LIN {X 0,Y 509.297,Z 394.262,A -85,B 0,C 180,E1 -5484.06,E2 -5484.06} C_VEL
LIN {X 0,Y 509.19,Z 398.581,A -85,B 0,C 180,E1 -5485.25,E2 -5485.25} C_VEL
LIN {X 0,Y 509.246,Z 400.946,A -85,B 0,C 180,E1 -5486.043,E2 -5486.043} C_VEL
LIN {X 0,Y 509.201,Z 402.741,A -85,B 0,C 180,E1 -5486.835,E2 -5486.835} C_VEL
LIN {X 0,Y 509.113,Z 405.178,A -85,B 0,C 180,E1 -5488.418,E2 -5488.418} C_VEL
LIN {X 0,Y 509.076,Z 405.764,A -85,B 0,C 180,E1 -5489.209,E2 -5489.209} C_VEL
LIN {X 0,Y 509.076,Z 405.764,A -85,B 0,C 180,E1 -5490.791,E2 -5490.791} C_VEL
LIN {X 0,Y 509.113,Z 405.178,A -85,B 0,C 180,E1 -5491.582,E2 -5491.582} C_VEL
LIN {X 0,Y 509.201,Z 402.741,A -85,B 0,C 180,E1 -5493.165,E2 -5493.165} C_VEL
LIN {X 0,Y 509.206,Z 399.797,A -85,B 0,C 180,E1 -5494.353,E2 -5494.353} C_VEL
LIN {X 0,Y 509.283,Z 395.815,A -85,B 0,C 180,E1 -5495.543,E2 -5495.543} C_VEL
LIN {X 0,Y 509.305,Z 390.878,A -85,B 0,C 180,E1 -5496.696,E2 -5496.696} C_VEL
LIN {X 0,Y 509.461,Z 385.428,A -85,B 0,C 180,E1 -5497.73,E2 -5497.73} C_VEL
LIN {X 0,Y 509.641,Z 379.112,A -85,B 0,C 180,E1 -5498.725,E2 -5498.725} C_VEL
LIN {X 0,Y 509.831,Z 373.161,A -85,B 0,C 180,E1 -5499.521,E2 -5499.521} C_VEL
LIN {X 0,Y 509.999,Z 366.231,A -85,B 0,C 180,E1 -5500.32,E2 -5500.32} C_VEL
LIN {X 0,Y 510.309,Z 358.051,A -85,B 0,C 180,E1 -5501.117,E2 -5501.117} C_VEL
LIN {X 0,Y 510.555,Z 349.536,A -85,B 0,C 180,E1 -5501.815,E2 -5501.815} C_VEL
LIN {X 0,Y 510.838,Z 339.999,A -85,B 0,C 180,E1 -5502.464,E2 -5502.464} C_VEL
LIN {X 0,Y 511.107,Z 330.048,A -85,B 0,C 180,E1 -5503.012,E2 -5503.012} C_VEL
LIN {X 0,Y 511.372,Z 319.682,A -85,B 0,C 180,E1 -5503.461,E2 -5503.461} C_VEL
LIN {X 0,Y 511.591,Z 308.831,A -85,B 0,C 180,E1 -5503.809,E2 -5503.809} C_VEL
LIN {X 0,Y 511.838,Z 295.749,A -85,B 0,C 180,E1 -5504.081,E2 -5504.081} C_VEL
LIN {X 0,Y 512.093,Z 207.59,A -85,B 0,C 180,E1 -5505.325,E2 -5505.325} C_VEL
LIN {X 0,Y 510.014,Z 195.134,A -85,B 0,C 180,E1 -5505.587,E2 -5505.587} C_VEL
LIN {X 0,Y 510.036,Z 192.862,A -85,B 0,C 180,E1 -5505.997,E2 -5505.997} C_VEL
LIN {X 0,Y 510.351,Z 179.568,A -85,B 0,C 180,E1 -5508.673,E2 -5508.673} C_VEL
LIN {X 0,Y 510.701,Z 165.975,A -85,B 0,C 180,E1 -5511.388,E2 -5511.388} C_VEL
LIN {X 0,Y 511.205,Z 151.526,A -85,B 0,C 180,E1 -5514.358,E2 -5514.358} C_VEL
LIN {X 0,Y 510.606,Z 146.371,A -85,B 0,C 180,E1 -5515.475,E2 -5515.475} C_VEL
LIN {X 0,Y 509.929,Z 142.498,A -85,B 0,C 180,E1 -5516.381,E2 -5516.381} C_VEL
LIN {X 0,Y 509.875,Z 142.472,A -85,B 0,C 180,E1 -5518.844,E2 -5518.844} C_VEL
LIN {X 0,Y 509.822,Z 142.482,A -85,B 0,C 180,E1 -5521.59,E2 -5521.59} C_VEL
LIN {X 0,Y 509.848,Z 142.473,A -85,B 0,C 180,E1 -5524.413,E2 -5524.413} C_VEL
LIN {X 0,Y 509.818,Z 142.478,A -85,B 0,C 180,E1 -5527.34,E2 -5527.34} C_VEL
LIN {X 0,Y 509.838,Z 142.466,A -85,B 0,C 180,E1 -5530.382,E2 -5530.382} C_VEL
LIN {X 0,Y 509.822,Z 142.477,A -85,B 0,C 180,E1 -5533.062,E2 -5533.062} C_VEL
LIN {X 0,Y 509.822,Z 142.48,A -85,B 0,C 180,E1 -5535.793,E2 -5535.793} C_VEL
LIN {X 0,Y 509.854,Z 142.471,A -85,B 0,C 180,E1 -5538.574,E2 -5538.574} C_VEL
LIN {X 0,Y 509.849,Z 142.475,A -85,B 0,C 180,E1 -5541.786,E2 -5541.786} C_VEL
LIN {X 0,Y 509.831,Z 142.473,A -85,B 0,C 180,E1 -5544.622,E2 -5544.622} C_VEL
LIN {X 0,Y 509.862,Z 142.475,A -85,B 0,C 180,E1 -5547.48,E2 -5547.48} C_VEL
LIN {X 0,Y 509.857,Z 142.47,A -85,B 0,C 180,E1 -5550.273,E2 -5550.273} C_VEL
LIN {X 0,Y 509.882,Z 142.466,A -85,B 0,C 180,E1 -5552.944,E2 -5552.944} C_VEL
LIN {X 0,Y 509.862,Z 142.471,A -85,B 0,C 180,E1 -5555.573,E2 -5555.573} C_VEL
LIN {X 0,Y 509.848,Z 142.474,A -85,B 0,C 180,E1 -5558.998,E2 -5558.998} C_VEL
LIN {X 0,Y 509.886,Z 142.458,A -85,B 0,C 180,E1 -5561.999,E2 -5561.999} C_VEL
LIN {X 0,Y 509.908,Z 142.471,A -85,B 0,C 180,E1 -5564.818,E2 -5564.818} C_VEL
LIN {X 0,Y 509.897,Z 142.464,A -85,B 0,C 180,E1 -5568.124,E2 -5568.124} C_VEL
LIN {X 0,Y 509.911,Z 142.457,A -85,B 0,C 180,E1 -5571.279,E2 -5571.279} C_VEL
LIN {X 0,Y 509.975,Z 142.454,A -85,B 0,C 180,E1 -5573.67,E2 -5573.67} C_VEL
LIN {X 0,Y 510.051,Z 142.444,A -85,B 0,C 180,E1 -5577.63,E2 -5577.63} C_VEL
LIN {X 0,Y 510.06,Z 142.44,A -85,B 0,C 180,E1 -5580.789,E2 -5580.789} C_VEL
LIN {X 0,Y 509.952,Z 142.457,A -85,B 0,C 180,E1 -5583.16,E2 -5583.16} C_VEL
LIN {X 0,Y 509.974,Z 142.46,A -85,B 0,C 180,E1 -5586.329,E2 -5586.329} C_VEL
LIN {X 0,Y 509.911,Z 142.456,A -85,B 0,C 180,E1 -5588.72,E2 -5588.72} C_VEL
LIN {X 0,Y 509.9,Z 142.465,A -85,B 0,C 180,E1 -5591.931,E2 -5591.931} C_VEL
LIN {X 0,Y 509.889,Z 142.467,A -85,B 0,C 180,E1 -5595.241,E2 -5595.241} C_VEL
LIN {X 0,Y 509.884,Z 142.464,A -85,B 0,C 180,E1 -5598.001,E2 -5598.001} C_VEL
LIN {X 0,Y 509.845,Z 142.468,A -85,B 0,C 180,E1 -5601.001,E2 -5601.001} C_VEL
LIN {X 0,Y 509.832,Z 142.479,A -85,B 0,C 180,E1 -5603.563,E2 -5603.563} C_VEL
LIN {X 0,Y 509.909,Z 142.458,A -85,B 0,C 180,E1 -5606.379,E2 -5606.379} C_VEL
LIN {X 0,Y 509.872,Z 142.465,A -85,B 0,C 180,E1 -5608.844,E2 -5608.844} C_VEL
LIN {X 0,Y 509.821,Z 142.482,A -85,B 0,C 180,E1 -5611.589,E2 -5611.589} C_VEL
LIN {X 0,Y 509.85,Z 142.464,A -85,B 0,C 180,E1 -5614.413,E2 -5614.413} C_VEL
LIN {X 0,Y 509.814,Z 142.483,A -85,B 0,C 180,E1 -5617.34,E2 -5617.34} C_VEL
LIN {X 0,Y 509.833,Z 142.469,A -85,B 0,C 180,E1 -5620.382,E2 -5620.382} C_VEL
LIN {X 0,Y 509.836,Z 142.479,A -85,B 0,C 180,E1 -5623.064,E2 -5623.064} C_VEL
LIN {X 0,Y 509.825,Z 142.469,A -85,B 0,C 180,E1 -5625.792,E2 -5625.792} C_VEL
LIN {X 0,Y 509.853,Z 142.457,A -85,B 0,C 180,E1 -5628.575,E2 -5628.575} C_VEL
LIN {X 0,Y 509.847,Z 142.473,A -85,B 0,C 180,E1 -5631.786,E2 -5631.786} C_VEL
LIN {X 0,Y 509.827,Z 142.471,A -85,B 0,C 180,E1 -5633.729,E2 -5633.729} C_VEL
LIN {X 0,Y 509.161,Z 142.556,A -85,B 0,C 180,E1 -5634.388,E2 -5634.388} C_VEL
LIN {X 0,Y 506.344,Z 142.91,A -85,B 0,C 180,E1 -5635.46,E2 -5635.46} C_VEL
LIN {X 0,Y 503.952,Z 143.211,A -85,B 0,C 180,E1 -5636.324,E2 -5636.324} C_VEL
LIN {X 0,Y 502.903,Z 143.341,A -85,B 0,C 180,E1 -5636.99,E2 -5636.99} C_VEL
LIN {X 0,Y 502.806,Z 143.351,A -85,B 0,C 180,E1 -5637.216,E2 -5637.216} C_VEL
LIN {X 0,Y 502.826,Z 143.344,A -85,B 0,C 180,E1 -5640.062,E2 -5640.062} C_VEL
LIN {X 0,Y 502.83,Z 143.351,A -85,B 0,C 180,E1 -5642.533,E2 -5642.533} C_VEL
LIN {X 0,Y 502.825,Z 143.349,A -85,B 0,C 180,E1 -5645.299,E2 -5645.299} C_VEL
LIN {X 0,Y 502.781,Z 143.354,A -85,B 0,C 180,E1 -5647.827,E2 -5647.827} C_VEL
LIN {X 0,Y 502.822,Z 143.355,A -85,B 0,C 180,E1 -5650.4,E2 -5650.4} C_VEL
LIN {X 0,Y 502.83,Z 143.35,A -85,B 0,C 180,E1 -5652.932,E2 -5652.932} C_VEL
LIN {X 0,Y 502.842,Z 143.347,A -85,B 0,C 180,E1 -5655.429,E2 -5655.429} C_VEL
LIN {X 0,Y 502.874,Z 143.346,A -85,B 0,C 180,E1 -5658.717,E2 -5658.717} C_VEL
LIN {X 0,Y 502.899,Z 143.344,A -85,B 0,C 180,E1 -5661.967,E2 -5661.967} C_VEL
LIN {X 0,Y 502.936,Z 143.34,A -85,B 0,C 180,E1 -5664.387,E2 -5664.387} C_VEL
LIN {X 0,Y 503.023,Z 143.327,A -85,B 0,C 180,E1 -5667.598,E2 -5667.598} C_VEL
LIN {X 0,Y 503.025,Z 143.33,A -85,B 0,C 180,E1 -5670,E2 -5670} C_VEL
LIN {X 0,Y 503.023,Z 143.327,A -85,B 0,C 180,E1 -5672.402,E2 -5672.402} C_VEL
LIN {X 0,Y 502.936,Z 143.34,A -85,B 0,C 180,E1 -5675.613,E2 -5675.613} C_VEL
LIN {X 0,Y 502.899,Z 143.344,A -85,B 0,C 180,E1 -5678.033,E2 -5678.033} C_VEL
LIN {X 0,Y 502.874,Z 143.346,A -85,B 0,C 180,E1 -5681.283,E2 -5681.283} C_VEL
LIN {X 0,Y 502.842,Z 143.347,A -85,B 0,C 180,E1 -5684.571,E2 -5684.571} C_VEL
LIN {X 0,Y 502.858,Z 143.348,A -85,B 0,C 180,E1 -5687.907,E2 -5687.907} C_VEL
LIN {X 0,Y 502.825,Z 143.349,A -85,B 0,C 180,E1 -5690.536,E2 -5690.536} C_VEL
LIN {X 0,Y 502.793,Z 143.356,A -85,B 0,C 180,E1 -5693.04,E2 -5693.04} C_VEL
LIN {X 0,Y 502.836,Z 143.35,A -85,B 0,C 180,E1 -5695.675,E2 -5695.675} C_VEL
LIN {X 0,Y 502.838,Z 143.344,A -85,B 0,C 180,E1 -5698.372,E2 -5698.372} C_VEL
LIN {X 0,Y 502.793,Z 143.355,A -85,B 0,C 180,E1 -5701.5,E2 -5701.5} C_VEL
LIN {X 0,Y 502.8,Z 143.343,A -85,B 0,C 180,E1 -5704.444,E2 -5704.444} C_VEL
LIN {X 0,Y 502.776,Z 143.36,A -85,B 0,C 180,E1 -5707.178,E2 -5707.178} C_VEL
LIN {X 0,Y 502.783,Z 143.348,A -85,B 0,C 180,E1 -5710.015,E2 -5710.015} C_VEL
LIN {X 0,Y 502.797,Z 143.334,A -85,B 0,C 180,E1 -5712.199,E2 -5712.199} C_VEL
LIN {X 0,Y 502.796,Z 143.351,A -85,B 0,C 180,E1 -5715.468,E2 -5715.468} C_VEL
LIN {X 0,Y 502.825,Z 143.346,A -85,B 0,C 180,E1 -5717.864,E2 -5717.864} C_VEL
LIN {X 0,Y 502.797,Z 143.354,A -85,B 0,C 180,E1 -5721.024,E2 -5721.024} C_VEL
LIN {X 0,Y 502.781,Z 143.355,A -85,B 0,C 180,E1 -5724.167,E2 -5724.167} C_VEL
LIN {X 0,Y 502.828,Z 143.347,A -85,B 0,C 180,E1 -5726.993,E2 -5726.993} C_VEL
LIN {X 0,Y 502.809,Z 143.353,A -85,B 0,C 180,E1 -5730.065,E2 -5730.065} C_VEL
LIN {X 0,Y 502.831,Z 143.343,A -85,B 0,C 180,E1 -5732.534,E2 -5732.534} C_VEL
LIN {X 0,Y 502.824,Z 143.346,A -85,B 0,C 180,E1 -5735.299,E2 -5735.299} C_VEL
LIN {X 0,Y 502.78,Z 143.356,A -85,B 0,C 180,E1 -5737.827,E2 -5737.827} C_VEL
LIN {X 0,Y 502.821,Z 143.34,A -85,B 0,C 180,E1 -5740.401,E2 -5740.401} C_VEL
LIN {X 0,Y 502.829,Z 143.343,A -85,B 0,C 180,E1 -5742.932,E2 -5742.932} C_VEL
LIN {X 0,Y 502.841,Z 143.346,A -85,B 0,C 180,E1 -5745.43,E2 -5745.43} C_VEL
LIN {X 0,Y 502.873,Z 143.333,A -85,B 0,C 180,E1 -5748.717,E2 -5748.717} C_VEL
LIN {X 0,Y 502.897,Z 143.339,A -85,B 0,C 180,E1 -5751.967,E2 -5751.967} C_VEL
LIN {X 0,Y 502.934,Z 143.334,A -85,B 0,C 180,E1 -5754.387,E2 -5754.387} C_VEL
LIN {X 0,Y 503.02,Z 143.325,A -85,B 0,C 180,E1 -5757.598,E2 -5757.598} C_VEL
LIN {X 0,Y 503.024,Z 143.315,A -85,B 0,C 180,E1 -5760,E2 -5760} C_VEL
LIN {X 0,Y 503.021,Z 143.319,A -85,B 0,C 180,E1 -5762.403,E2 -5762.403} C_VEL
LIN {X 0,Y 502.934,Z 143.338,A -85,B 0,C 180,E1 -5765.614,E2 -5765.614} C_VEL
LIN {X 0,Y 502.898,Z 143.331,A -85,B 0,C 180,E1 -5768.034,E2 -5768.034} C_VEL
LIN {X 0,Y 502.874,Z 143.338,A -85,B 0,C 180,E1 -5771.284,E2 -5771.284} C_VEL
LIN {X 0,Y 502.842,Z 143.344,A -85,B 0,C 180,E1 -5774.571,E2 -5774.571} C_VEL
LIN {X 0,Y 502.859,Z 143.333,A -85,B 0,C 180,E1 -5777.907,E2 -5777.907} C_VEL
LIN {X 0,Y 502.826,Z 143.342,A -85,B 0,C 180,E1 -5780.537,E2 -5780.537} C_VEL
LIN {X 0,Y 502.789,Z 143.358,A -85,B 0,C 180,E1 -5783.041,E2 -5783.041} C_VEL
LIN {X 0,Y 502.838,Z 143.339,A -85,B 0,C 180,E1 -5785.676,E2 -5785.676} C_VEL
LIN {X 0,Y 502.838,Z 143.341,A -85,B 0,C 180,E1 -5788.373,E2 -5788.373} C_VEL
LIN {X 0,Y 502.792,Z 143.351,A -85,B 0,C 180,E1 -5791.499,E2 -5791.499} C_VEL
LIN {X 0,Y 502.804,Z 143.344,A -85,B 0,C 180,E1 -5793.994,E2 -5793.994} C_VEL
LIN {X 0,Y 502.776,Z 143.355,A -85,B 0,C 180,E1 -5797.178,E2 -5797.178} C_VEL
LIN {X 0,Y 502.787,Z 143.35,A -85,B 0,C 180,E1 -5800.016,E2 -5800.016} C_VEL
LIN {X 0,Y 502.802,Z 143.353,A -85,B 0,C 180,E1 -5802.2,E2 -5802.2} C_VEL
LIN {X 0,Y 502.785,Z 143.351,A -85,B 0,C 180,E1 -5805.471,E2 -5805.471} C_VEL
LIN {X 0,Y 502.82,Z 143.341,A -85,B 0,C 180,E1 -5808.935,E2 -5808.935} C_VEL
LIN {X 0,Y 502.794,Z 143.355,A -85,B 0,C 180,E1 -5812.047,E2 -5812.047} C_VEL
LIN {X 0,Y 502.8,Z 143.349,A -85,B 0,C 180,E1 -5815.035,E2 -5815.035} C_VEL
LIN {X 0,Y 502.785,Z 143.354,A -85,B 0,C 180,E1 -5817.916,E2 -5817.916} C_VEL
LIN {X 0,Y 502.824,Z 143.351,A -85,B 0,C 180,E1 -5820.713,E2 -5820.713} C_VEL
LIN {X 0,Y 502.884,Z 143.391,A -85,B 0,C 180,E1 -5823.435,E2 -5823.435} C_VEL
LIN {X 0,Y 504.214,Z 151.389,A -85,B 0,C 180,E1 -5825.282,E2 -5825.282} C_VEL
LIN {X 0,Y 503.775,Z 164.795,A -85,B 0,C 180,E1 -5828.088,E2 -5828.088} C_VEL
LIN {X 0,Y 503.386,Z 178.303,A -85,B 0,C 180,E1 -5830.847,E2 -5830.847} C_VEL
LIN {X 0,Y 503.067,Z 190.691,A -85,B 0,C 180,E1 -5833.358,E2 -5833.358} C_VEL
LIN {X 0,Y 502.995,Z 194.737,A -85,B 0,C 180,E1 -5834.174,E2 -5834.174} C_VEL
LIN {X 0,Y 504.04,Z 201.188,A -85,B 0,C 180,E1 -5834.334,E2 -5834.334} C_VEL
LIN {X 0,Y 505.337,Z 210.355,A -85,B 0,C 180,E1 -5834.508,E2 -5834.508} C_VEL
LIN {X 0,Y 504.897,Z 299.619,A -85,B 0,C 180,E1 -5835.799,E2 -5835.799} C_VEL
LIN {X 0,Y 504.687,Z 309.514,A -85,B 0,C 180,E1 -5836.024,E2 -5836.024} C_VEL
LIN {X 0,Y 504.474,Z 319.491,A -85,B 0,C 180,E1 -5836.352,E2 -5836.352} C_VEL
LIN {X 0,Y 504.15,Z 329.855,A -85,B 0,C 180,E1 -5836.805,E2 -5836.805} C_VEL
LIN {X 0,Y 503.88,Z 339.867,A -85,B 0,C 180,E1 -5837.365,E2 -5837.365} C_VEL
LIN {X 0,Y 503.623,Z 347.992,A -85,B 0,C 180,E1 -5837.917,E2 -5837.917} C_VEL
LIN {X 0,Y 503.309,Z 356.722,A -85,B 0,C 180,E1 -5838.625,E2 -5838.625} C_VEL
LIN {X 0,Y 503.069,Z 364.119,A -85,B 0,C 180,E1 -5839.333,E2 -5839.333} C_VEL
LIN {X 0,Y 502.848,Z 371.341,A -85,B 0,C 180,E1 -5840.142,E2 -5840.142} C_VEL
LIN {X 0,Y 502.631,Z 377.543,A -85,B 0,C 180,E1 -5840.95,E2 -5840.95} C_VEL
LIN {X 0,Y 502.427,Z 384.08,A -85,B 0,C 180,E1 -5841.959,E2 -5841.959} C_VEL
LIN {X 0,Y 502.274,Z 389.633,A -85,B 0,C 180,E1 -5842.988,E2 -5842.988} C_VEL
LIN {X 0,Y 502.2,Z 394.069,A -85,B 0,C 180,E1 -5843.975,E2 -5843.975} C_VEL
LIN {X 0,Y 502.112,Z 398.389,A -85,B 0,C 180,E1 -5845.183,E2 -5845.183} C_VEL
LIN {X 0,Y 502.139,Z 400.754,A -85,B 0,C 180,E1 -5845.987,E2 -5845.987} C_VEL
LIN {X 0,Y 502.12,Z 402.549,A -85,B 0,C 180,E1 -5846.791,E2 -5846.791} C_VEL
LIN {X 0,Y 502.036,Z 404.987,A -85,B 0,C 180,E1 -5848.396,E2 -5848.396} C_VEL
LIN {X 0,Y 501.993,Z 405.573,A -85,B 0,C 180,E1 -5849.198,E2 -5849.198} C_VEL
LIN {X 0,Y 501.993,Z 405.573,A -85,B 0,C 180,E1 -5850.802,E2 -5850.802} C_VEL
LIN {X 0,Y 502.036,Z 404.987,A -85,B 0,C 180,E1 -5851.604,E2 -5851.604} C_VEL
LIN {X 0,Y 502.12,Z 402.549,A -85,B 0,C 180,E1 -5853.209,E2 -5853.209} C_VEL
LIN {X 0,Y 502.104,Z 399.604,A -85,B 0,C 180,E1 -5854.415,E2 -5854.415} C_VEL
LIN {X 0,Y 502.199,Z 395.622,A -85,B 0,C 180,E1 -5855.622,E2 -5855.622} C_VEL
LIN {X 0,Y 502.217,Z 390.686,A -85,B 0,C 180,E1 -5856.791,E2 -5856.791} C_VEL
LIN {X 0,Y 502.384,Z 385.235,A -85,B 0,C 180,E1 -5857.839,E2 -5857.839} C_VEL
LIN {X 0,Y 502.58,Z 378.919,A -85,B 0,C 180,E1 -5858.848,E2 -5858.848} C_VEL
LIN {X 0,Y 502.789,Z 372.968,A -85,B 0,C 180,E1 -5859.656,E2 -5859.656} C_VEL
LIN {X 0,Y 502.979,Z 366.038,A -85,B 0,C 180,E1 -5860.466,E2 -5860.466} C_VEL
LIN {X 0,Y 503.27,Z 357.857,A -85,B 0,C 180,E1 -5861.274,E2 -5861.274} C_VEL
LIN {X 0,Y 503.556,Z 349.343,A -85,B 0,C 180,E1 -5861.982,E2 -5861.982} C_VEL
LIN {X 0,Y 503.869,Z 340.259,A -85,B 0,C 180,E1 -5862.611,E2 -5862.611} C_VEL
LIN {X 0,Y 504.145,Z 330.863,A -85,B 0,C 180,E1 -5863.144,E2 -5863.144} C_VEL
LIN {X 0,Y 504.427,Z 320.779,A -85,B 0,C 180,E1 -5863.598,E2 -5863.598} C_VEL
LIN {X 0,Y 504.664,Z 311.263,A -85,B 0,C 180,E1 -5863.925,E2 -5863.925} C_VEL
LIN {X 0,Y 504.854,Z 300.95,A -85,B 0,C 180,E1 -5864.177,E2 -5864.177} C_VEL
LIN {X 0,Y 505.149,Z 245.451,A -85,B 0,C 180,E1 -5864.992,E2 -5864.992} C_VEL
LIN {X 0,Y 505.146,Z 207.814,A -85,B 0,C 180,E1 -5865.535,E2 -5865.535} C_VEL
LIN {X 0,Y 502.988,Z 195.087,A -85,B 0,C 180,E1 -5865.803,E2 -5865.803} C_VEL
LIN {X 0,Y 502.966,Z 193.979,A -85,B 0,C 180,E1 -5865.947,E2 -5865.947} C_VEL
LIN {X 0,Y 503.352,Z 180.482,A -85,B 0,C 180,E1 -5868.731,E2 -5868.731} C_VEL
LIN {X 0,Y 503.708,Z 166.888,A -85,B 0,C 180,E1 -5871.485,E2 -5871.485} C_VEL
LIN {X 0,Y 504.223,Z 153.482,A -85,B 0,C 180,E1 -5874.279,E2 -5874.279} C_VEL
LIN {X 0,Y 503.896,Z 148.963,A -85,B 0,C 180,E1 -5875.26,E2 -5875.26} C_VEL
LIN {X 0,Y 502.884,Z 143.372,A -85,B 0,C 180,E1 -5876.565,E2 -5876.565} C_VEL
LIN {X 0,Y 502.824,Z 143.351,A -85,B 0,C 180,E1 -5879.287,E2 -5879.287} C_VEL
LIN {X 0,Y 502.785,Z 143.355,A -85,B 0,C 180,E1 -5882.084,E2 -5882.084} C_VEL
LIN {X 0,Y 502.8,Z 143.349,A -85,B 0,C 180,E1 -5884.965,E2 -5884.965} C_VEL
LIN {X 0,Y 502.794,Z 143.355,A -85,B 0,C 180,E1 -5887.953,E2 -5887.953} C_VEL
LIN {X 0,Y 502.82,Z 143.341,A -85,B 0,C 180,E1 -5891.065,E2 -5891.065} C_VEL
LIN {X 0,Y 502.785,Z 143.351,A -85,B 0,C 180,E1 -5894.529,E2 -5894.529} C_VEL
LIN {X 0,Y 502.794,Z 143.354,A -85,B 0,C 180,E1 -5897.86,E2 -5897.86} C_VEL
LIN {X 0,Y 502.8,Z 143.349,A -85,B 0,C 180,E1 -5901.023,E2 -5901.023} C_VEL
LIN {X 0,Y 502.774,Z 143.351,A -85,B 0,C 180,E1 -5904.168,E2 -5904.168} C_VEL
LIN {X 0,Y 502.831,Z 143.344,A -85,B 0,C 180,E1 -5906.993,E2 -5906.993} C_VEL
LIN {X 0,Y 502.813,Z 143.348,A -85,B 0,C 180,E1 -5910.064,E2 -5910.064} C_VEL
LIN {X 0,Y 502.83,Z 143.342,A -85,B 0,C 180,E1 -5912.533,E2 -5912.533} C_VEL
LIN {X 0,Y 502.825,Z 143.35,A -85,B 0,C 180,E1 -5915.299,E2 -5915.299} C_VEL
LIN {X 0,Y 502.777,Z 143.351,A -85,B 0,C 180,E1 -5917.826,E2 -5917.826} C_VEL
LIN {X 0,Y 502.823,Z 143.343,A -85,B 0,C 180,E1 -5920.4,E2 -5920.4} C_VEL
LIN {X 0,Y 502.832,Z 143.347,A -85,B 0,C 180,E1 -5922.931,E2 -5922.931} C_VEL
LIN {X 0,Y 502.842,Z 143.344,A -85,B 0,C 180,E1 -5925.429,E2 -5925.429} C_VEL
LIN {X 0,Y 502.874,Z 143.338,A -85,B 0,C 180,E1 -5928.716,E2 -5928.716} C_VEL
LIN {X 0,Y 502.898,Z 143.331,A -85,B 0,C 180,E1 -5931.966,E2 -5931.966} C_VEL
LIN {X 0,Y 502.934,Z 143.338,A -85,B 0,C 180,E1 -5934.386,E2 -5934.386} C_VEL
LIN {X 0,Y 503.021,Z 143.319,A -85,B 0,C 180,E1 -5937.597,E2 -5937.597} C_VEL
LIN {X 0,Y 503.024,Z 143.315,A -85,B 0,C 180,E1 -5940,E2 -5940} C_VEL
LIN {X 0,Y 503.02,Z 143.325,A -85,B 0,C 180,E1 -5942.402,E2 -5942.402} C_VEL
LIN {X 0,Y 502.934,Z 143.334,A -85,B 0,C 180,E1 -5945.613,E2 -5945.613} C_VEL
LIN {X 0,Y 502.897,Z 143.339,A -85,B 0,C 180,E1 -5948.033,E2 -5948.033} C_VEL
LIN {X 0,Y 502.873,Z 143.333,A -85,B 0,C 180,E1 -5951.283,E2 -5951.283} C_VEL
LIN {X 0,Y 502.841,Z 143.346,A -85,B 0,C 180,E1 -5954.57,E2 -5954.57} C_VEL
LIN {X 0,Y 502.857,Z 143.34,A -85,B 0,C 180,E1 -5957.907,E2 -5957.907} C_VEL
LIN {X 0,Y 502.824,Z 143.343,A -85,B 0,C 180,E1 -5960.536,E2 -5960.536} C_VEL
LIN {X 0,Y 502.792,Z 143.351,A -85,B 0,C 180,E1 -5963.04,E2 -5963.04} C_VEL
LIN {X 0,Y 502.837,Z 143.347,A -85,B 0,C 180,E1 -5965.675,E2 -5965.675} C_VEL
LIN {X 0,Y 502.836,Z 143.342,A -85,B 0,C 180,E1 -5968.372,E2 -5968.372} C_VEL
LIN {X 0,Y 502.792,Z 143.359,A -85,B 0,C 180,E1 -5971.499,E2 -5971.499} C_VEL
LIN {X 0,Y 502.802,Z 143.341,A -85,B 0,C 180,E1 -5974.445,E2 -5974.445} C_VEL
LIN {X 0,Y 502.776,Z 143.358,A -85,B 0,C 180,E1 -5977.178,E2 -5977.178} C_VEL
LIN {X 0,Y 502.783,Z 143.348,A -85,B 0,C 180,E1 -5980.015,E2 -5980.015} C_VEL
LIN {X 0,Y 502.798,Z 143.349,A -85,B 0,C 180,E1 -5982.199,E2 -5982.199} C_VEL
LIN {X 0,Y 502.795,Z 143.348,A -85,B 0,C 180,E1 -5985.468,E2 -5985.468} C_VEL
LIN {X 0,Y 502.815,Z 143.337,A -85,B 0,C 180,E1 -5988.934,E2 -5988.934} C_VEL
LIN {X 0,Y 502.79,Z 143.352,A -85,B 0,C 180,E1 -5992.046,E2 -5992.046} C_VEL
LIN {X 0,Y 502.805,Z 143.344,A -85,B 0,C 180,E1 -5995.035,E2 -5995.035} C_VEL
LIN {X 0,Y 502.806,Z 143.351,A -85,B 0,C 180,E1 -5997.216,E2 -5997.216} C_VEL
LIN {X 0,Y 502.107,Z 143.437,A -85,B 0,C 180,E1 -5997.884,E2 -5997.884} C_VEL
LIN {X 0,Y 499.249,Z 143.796,A -85,B 0,C 180,E1 -5998.97,E2 -5998.97} C_VEL
LIN {X 0,Y 496.858,Z 144.09,A -85,B 0,C 180,E1 -5999.845,E2 -5999.845} C_VEL
LIN {X 0,Y 495.839,Z 144.216,A -85,B 0,C 180,E1 -6000.521,E2 -6000.521} C_VEL
LIN {X 0,Y 495.759,Z 144.225,A -85,B 0,C 180,E1 -6000.75,E2 -6000.75} C_VEL
LIN {X 0,Y 495.787,Z 144.225,A -85,B 0,C 180,E1 -6003.932,E2 -6003.932} C_VEL
LIN {X 0,Y 495.762,Z 144.23,A -85,B 0,C 180,E1 -6007.138,E2 -6007.138} C_VEL
LIN {X 0,Y 495.774,Z 144.23,A -85,B 0,C 180,E1 -6010.11,E2 -6010.11} C_VEL
LIN {X 0,Y 495.783,Z 144.231,A -85,B 0,C 180,E1 -6012.682,E2 -6012.682} C_VEL
LIN {X 0,Y 495.787,Z 144.226,A -85,B 0,C 180,E1 -6015.217,E2 -6015.217} C_VEL
LIN {X 0,Y 495.849,Z 144.223,A -85,B 0,C 180,E1 -6018.555,E2 -6018.555} C_VEL
LIN {X 0,Y 495.87,Z 144.22,A -85,B 0,C 180,E1 -6021.852,E2 -6021.852} C_VEL
LIN {X 0,Y 495.894,Z 144.218,A -85,B 0,C 180,E1 -6024.307,E2 -6024.307} C_VEL
LIN {X 0,Y 495.991,Z 144.203,A -85,B 0,C 180,E1 -6027.564,E2 -6027.564} C_VEL
LIN {X 0,Y 495.996,Z 144.206,A -85,B 0,C 180,E1 -6030,E2 -6030} C_VEL
LIN {X 0,Y 495.992,Z 144.203,A -85,B 0,C 180,E1 -6032.436,E2 -6032.436} C_VEL
LIN {X 0,Y 495.894,Z 144.218,A -85,B 0,C 180,E1 -6035.693,E2 -6035.693} C_VEL
LIN {X 0,Y 495.87,Z 144.22,A -85,B 0,C 180,E1 -6038.148,E2 -6038.148} C_VEL
LIN {X 0,Y 495.849,Z 144.223,A -85,B 0,C 180,E1 -6041.445,E2 -6041.445} C_VEL
LIN {X 0,Y 495.787,Z 144.226,A -85,B 0,C 180,E1 -6044.783,E2 -6044.783} C_VEL
LIN {X 0,Y 495.783,Z 144.231,A -85,B 0,C 180,E1 -6047.319,E2 -6047.319} C_VEL
LIN {X 0,Y 495.774,Z 144.23,A -85,B 0,C 180,E1 -6049.89,E2 -6049.89} C_VEL
LIN {X 0,Y 495.762,Z 144.23,A -85,B 0,C 180,E1 -6052.862,E2 -6052.862} C_VEL
LIN {X 0,Y 495.787,Z 144.225,A -85,B 0,C 180,E1 -6056.068,E2 -6056.068} C_VEL
LIN {X 0,Y 495.777,Z 144.225,A -85,B 0,C 180,E1 -6058.814,E2 -6058.814} C_VEL
LIN {X 0,Y 495.755,Z 144.23,A -85,B 0,C 180,E1 -6061.726,E2 -6061.726} C_VEL
LIN {X 0,Y 495.77,Z 144.219,A -85,B 0,C 180,E1 -6064.695,E2 -6064.695} C_VEL
LIN {X 0,Y 495.727,Z 144.234,A -85,B 0,C 180,E1 -6067.561,E2 -6067.561} C_VEL
LIN {X 0,Y 495.762,Z 144.221,A -85,B 0,C 180,E1 -6070.7,E2 -6070.7} C_VEL
LIN {X 0,Y 495.729,Z 144.223,A -85,B 0,C 180,E1 -6074.001,E2 -6074.001} C_VEL
LIN {X 0,Y 495.729,Z 144.233,A -85,B 0,C 180,E1 -6077.118,E2 -6077.118} C_VEL
LIN {X 0,Y 495.754,Z 144.223,A -85,B 0,C 180,E1 -6079.953,E2 -6079.953} C_VEL
LIN {X 0,Y 495.726,Z 144.239,A -85,B 0,C 180,E1 -6082.553,E2 -6082.553} C_VEL
LIN {X 0,Y 495.781,Z 144.216,A -85,B 0,C 180,E1 -6085.458,E2 -6085.458} C_VEL
LIN {X 0,Y 495.754,Z 144.234,A -85,B 0,C 180,E1 -6088.364,E2 -6088.364} C_VEL
LIN {X 0,Y 495.783,Z 144.22,A -85,B 0,C 180,E1 -6091.507,E2 -6091.507} C_VEL
LIN {X 0,Y 495.794,Z 144.218,A -85,B 0,C 180,E1 -6093.933,E2 -6093.933} C_VEL
LIN {X 0,Y 495.761,Z 144.227,A -85,B 0,C 180,E1 -6097.138,E2 -6097.138} C_VEL
LIN {X 0,Y 495.767,Z 144.222,A -85,B 0,C 180,E1 -6100.11,E2 -6100.11} C_VEL
LIN {X 0,Y 495.782,Z 144.222,A -85,B 0,C 180,E1 -6102.682,E2 -6102.682} C_VEL
LIN {X 0,Y 495.786,Z 144.224,A -85,B 0,C 180,E1 -6105.218,E2 -6105.218} C_VEL
LIN {X 0,Y 495.847,Z 144.209,A -85,B 0,C 180,E1 -6108.555,E2 -6108.555} C_VEL
LIN {X 0,Y 495.869,Z 144.212,A -85,B 0,C 180,E1 -6111.852,E2 -6111.852} C_VEL
LIN {X 0,Y 495.891,Z 144.212,A -85,B 0,C 180,E1 -6114.307,E2 -6114.307} C_VEL
LIN {X 0,Y 495.989,Z 144.201,A -85,B 0,C 180,E1 -6117.564,E2 -6117.564} C_VEL
LIN {X 0,Y 495.995,Z 144.19,A -85,B 0,C 180,E1 -6120,E2 -6120} C_VEL
LIN {X 0,Y 495.99,Z 144.195,A -85,B 0,C 180,E1 -6122.437,E2 -6122.437} C_VEL
LIN {X 0,Y 495.892,Z 144.214,A -85,B 0,C 180,E1 -6125.694,E2 -6125.694} C_VEL
LIN {X 0,Y 495.869,Z 144.205,A -85,B 0,C 180,E1 -6128.148,E2 -6128.148} C_VEL
LIN {X 0,Y 495.848,Z 144.216,A -85,B 0,C 180,E1 -6131.446,E2 -6131.446} C_VEL
LIN {X 0,Y 495.787,Z 144.225,A -85,B 0,C 180,E1 -6134.783,E2 -6134.783} C_VEL
LIN {X 0,Y 495.784,Z 144.219,A -85,B 0,C 180,E1 -6137.319,E2 -6137.319} C_VEL
LIN {X 0,Y 495.769,Z 144.219,A -85,B 0,C 180,E1 -6139.891,E2 -6139.891} C_VEL
LIN {X 0,Y 495.757,Z 144.232,A -85,B 0,C 180,E1 -6142.861,E2 -6142.861} C_VEL
LIN {X 0,Y 495.788,Z 144.217,A -85,B 0,C 180,E1 -6146.068,E2 -6146.068} C_VEL
LIN {X 0,Y 495.77,Z 144.227,A -85,B 0,C 180,E1 -6148.815,E2 -6148.815} C_VEL
LIN {X 0,Y 495.755,Z 144.227,A -85,B 0,C 180,E1 -6151.726,E2 -6151.726} C_VEL
LIN {X 0,Y 495.769,Z 144.225,A -85,B 0,C 180,E1 -6154.695,E2 -6154.695} C_VEL
LIN {X 0,Y 495.727,Z 144.231,A -85,B 0,C 180,E1 -6157.562,E2 -6157.562} C_VEL
LIN {X 0,Y 495.765,Z 144.23,A -85,B 0,C 180,E1 -6160.7,E2 -6160.7} C_VEL
LIN {X 0,Y 495.727,Z 144.233,A -85,B 0,C 180,E1 -6164.002,E2 -6164.002} C_VEL
LIN {X 0,Y 495.725,Z 144.232,A -85,B 0,C 180,E1 -6167.117,E2 -6167.117} C_VEL
LIN {X 0,Y 495.759,Z 144.221,A -85,B 0,C 180,E1 -6169.953,E2 -6169.953} C_VEL
LIN {X 0,Y 495.729,Z 144.235,A -85,B 0,C 180,E1 -6172.554,E2 -6172.554} C_VEL
LIN {X 0,Y 495.779,Z 144.224,A -85,B 0,C 180,E1 -6175.457,E2 -6175.457} C_VEL
LIN {X 0,Y 495.757,Z 144.232,A -85,B 0,C 180,E1 -6178.364,E2 -6178.364} C_VEL
LIN {X 0,Y 495.788,Z 144.23,A -85,B 0,C 180,E1 -6181.508,E2 -6181.508} C_VEL
LIN {X 0,Y 495.826,Z 144.276,A -85,B 0,C 180,E1 -6183.251,E2 -6183.251} C_VEL
LIN {X 0,Y 497.215,Z 152.315,A -85,B 0,C 180,E1 -6185.134,E2 -6185.134} C_VEL
LIN {X 0,Y 496.951,Z 161.806,A -85,B 0,C 180,E1 -6187.173,E2 -6187.173} C_VEL
LIN {X 0,Y 496.528,Z 176.073,A -85,B 0,C 180,E1 -6190.141,E2 -6190.141} C_VEL
LIN {X 0,Y 496.077,Z 190.529,A -85,B 0,C 180,E1 -6193.117,E2 -6193.117} C_VEL
LIN {X 0,Y 495.98,Z 194.514,A -85,B 0,C 180,E1 -6193.939,E2 -6193.939} C_VEL
LIN {X 0,Y 496.639,Z 198.909,A -85,B 0,C 180,E1 -6194.064,E2 -6194.064} C_VEL
LIN {X 0,Y 498.5,Z 211.149,A -85,B 0,C 180,E1 -6194.304,E2 -6194.304} C_VEL
LIN {X 0,Y 498.026,Z 299.428,A -85,B 0,C 180,E1 -6195.598,E2 -6195.598} C_VEL
LIN {X 0,Y 497.793,Z 310.197,A -85,B 0,C 180,E1 -6195.852,E2 -6195.852} C_VEL
LIN {X 0,Y 497.582,Z 319.3,A -85,B 0,C 180,E1 -6196.159,E2 -6196.159} C_VEL
LIN {X 0,Y 497.224,Z 329.663,A -85,B 0,C 180,E1 -6196.618,E2 -6196.618} C_VEL
LIN {X 0,Y 496.967,Z 338.879,A -85,B 0,C 180,E1 -6197.136,E2 -6197.136} C_VEL
LIN {X 0,Y 496.648,Z 347.799,A -85,B 0,C 180,E1 -6197.745,E2 -6197.745} C_VEL
LIN {X 0,Y 496.33,Z 356.53,A -85,B 0,C 180,E1 -6198.463,E2 -6198.463} C_VEL
LIN {X 0,Y 496.08,Z 363.927,A -85,B 0,C 180,E1 -6199.181,E2 -6199.181} C_VEL
LIN {X 0,Y 495.819,Z 371.148,A -85,B 0,C 180,E1 -6200.001,E2 -6200.001} C_VEL
LIN {X 0,Y 495.596,Z 377.351,A -85,B 0,C 180,E1 -6200.82,E2 -6200.82} C_VEL
LIN {X 0,Y 495.376,Z 383.887,A -85,B 0,C 180,E1 -6201.844,E2 -6201.844} C_VEL
LIN {X 0,Y 495.262,Z 388.389,A -85,B 0,C 180,E1 -6202.663,E2 -6202.663} C_VEL
LIN {X 0,Y 495.118,Z 393.416,A -85,B 0,C 180,E1 -6203.768,E2 -6203.768} C_VEL
LIN {X 0,Y 495.104,Z 396.96,A -85,B 0,C 180,E1 -6204.706,E2 -6204.706} C_VEL
LIN {X 0,Y 495.033,Z 400.562,A -85,B 0,C 180,E1 -6205.929,E2 -6205.929} C_VEL
LIN {X 0,Y 495.042,Z 402.358,A -85,B 0,C 180,E1 -6206.745,E2 -6206.745} C_VEL
LIN {X 0,Y 494.963,Z 404.796,A -85,B 0,C 180,E1 -6208.373,E2 -6208.373} C_VEL
LIN {X 0,Y 494.913,Z 405.382,A -85,B 0,C 180,E1 -6209.186,E2 -6209.186} C_VEL
LIN {X 0,Y 494.913,Z 405.382,A -85,B 0,C 180,E1 -6210.814,E2 -6210.814} C_VEL
LIN {X 0,Y 494.963,Z 404.796,A -85,B 0,C 180,E1 -6211.627,E2 -6211.627} C_VEL
LIN {X 0,Y 495.042,Z 402.358,A -85,B 0,C 180,E1 -6213.255,E2 -6213.255} C_VEL
LIN {X 0,Y 495.01,Z 399.412,A -85,B 0,C 180,E1 -6214.479,E2 -6214.479} C_VEL
LIN {X 0,Y 495.115,Z 395.43,A -85,B 0,C 180,E1 -6215.702,E2 -6215.702} C_VEL
LIN {X 0,Y 495.168,Z 390.302,A -85,B 0,C 180,E1 -6216.929,E2 -6216.929} C_VEL
LIN {X 0,Y 495.33,Z 385.043,A -85,B 0,C 180,E1 -6217.952,E2 -6217.952} C_VEL
LIN {X 0,Y 495.546,Z 378.727,A -85,B 0,C 180,E1 -6218.975,E2 -6218.975} C_VEL
LIN {X 0,Y 495.744,Z 372.775,A -85,B 0,C 180,E1 -6219.795,E2 -6219.795} C_VEL
LIN {X 0,Y 495.975,Z 365.846,A -85,B 0,C 180,E1 -6220.615,E2 -6220.615} C_VEL
LIN {X 0,Y 496.287,Z 357.665,A -85,B 0,C 180,E1 -6221.435,E2 -6221.435} C_VEL
LIN {X 0,Y 496.581,Z 349.151,A -85,B 0,C 180,E1 -6222.153,E2 -6222.153} C_VEL
LIN {X 0,Y 496.896,Z 340.546,A -85,B 0,C 180,E1 -6222.76,E2 -6222.76} C_VEL
LIN {X 0,Y 497.194,Z 330.67,A -85,B 0,C 180,E1 -6223.331,E2 -6223.331} C_VEL
LIN {X 0,Y 497.516,Z 321.876,A -85,B 0,C 180,E1 -6223.739,E2 -6223.739} C_VEL
LIN {X 0,Y 497.76,Z 311.946,A -85,B 0,C 180,E1 -6224.096,E2 -6224.096} C_VEL
LIN {X 0,Y 497.952,Z 302.09,A -85,B 0,C 180,E1 -6224.352,E2 -6224.352} C_VEL
LIN {X 0,Y 498.166,Z 279.271,A -85,B 0,C 180,E1 -6224.711,E2 -6224.711} C_VEL
LIN {X 0,Y 498.337,Z 208.885,A -85,B 0,C 180,E1 -6225.734,E2 -6225.734} C_VEL
LIN {X 0,Y 495.979,Z 194.756,A -85,B 0,C 180,E1 -6226.041,E2 -6226.041} C_VEL
LIN {X 0,Y 495.957,Z 193.457,A -85,B 0,C 180,E1 -6226.252,E2 -6226.252} C_VEL
LIN {X 0,Y 496.336,Z 182.061,A -85,B 0,C 180,E1 -6228.656,E2 -6228.656} C_VEL
LIN {X 0,Y 496.726,Z 167.802,A -85,B 0,C 180,E1 -6231.584,E2 -6231.584} C_VEL
LIN {X 0,Y 497.272,Z 154.381,A -85,B 0,C 180,E1 -6234.418,E2 -6234.418} C_VEL
LIN {X 0,Y 496.762,Z 149.257,A -85,B 0,C 180,E1 -6235.562,E2 -6235.562} C_VEL
LIN {X 0,Y 495.836,Z 144.249,A -85,B 0,C 180,E1 -6236.751,E2 -6236.751} C_VEL
LIN {X 0,Y 495.767,Z 144.229,A -85,B 0,C 180,E1 -6239.746,E2 -6239.746} C_VEL
LIN {X 0,Y 495.769,Z 144.227,A -85,B 0,C 180,E1 -6242.594,E2 -6242.594} C_VEL
LIN {X 0,Y 495.749,Z 144.228,A -85,B 0,C 180,E1 -6245.537,E2 -6245.537} C_VEL
LIN {X 0,Y 495.765,Z 144.225,A -85,B 0,C 180,E1 -6248.768,E2 -6248.768} C_VEL
LIN {X 0,Y 495.756,Z 144.23,A -85,B 0,C 180,E1 -6251.781,E2 -6251.781} C_VEL
LIN {X 0,Y 495.737,Z 144.232,A -85,B 0,C 180,E1 -6255.14,E2 -6255.14} C_VEL
LIN {X 0,Y 495.755,Z 144.228,A -85,B 0,C 180,E1 -6258.218,E2 -6258.218} C_VEL
LIN {X 0,Y 495.749,Z 144.233,A -85,B 0,C 180,E1 -6261.408,E2 -6261.408} C_VEL
LIN {X 0,Y 495.748,Z 144.226,A -85,B 0,C 180,E1 -6264.462,E2 -6264.462} C_VEL
LIN {X 0,Y 495.767,Z 144.231,A -85,B 0,C 180,E1 -6267.405,E2 -6267.405} C_VEL
LIN {X 0,Y 495.765,Z 144.226,A -85,B 0,C 180,E1 -6270.253,E2 -6270.253} C_VEL
LIN {X 0,Y 495.821,Z 144.216,A -85,B 0,C 180,E1 -6273.25,E2 -6273.25} C_VEL
LIN {X 0,Y 495.746,Z 144.228,A -85,B 0,C 180,E1 -6275.724,E2 -6275.724} C_VEL
LIN {X 0,Y 495.74,Z 144.229,A -85,B 0,C 180,E1 -6278.37,E2 -6278.37} C_VEL
LIN {X 0,Y 495.782,Z 144.218,A -85,B 0,C 180,E1 -6280.971,E2 -6280.971} C_VEL
LIN {X 0,Y 495.777,Z 144.222,A -85,B 0,C 180,E1 -6283.529,E2 -6283.529} C_VEL
LIN {X 0,Y 495.791,Z 144.223,A -85,B 0,C 180,E1 -6286.055,E2 -6286.055} C_VEL
LIN {X 0,Y 495.848,Z 144.216,A -85,B 0,C 180,E1 -6288.554,E2 -6288.554} C_VEL
LIN {X 0,Y 495.869,Z 144.205,A -85,B 0,C 180,E1 -6291.852,E2 -6291.852} C_VEL
LIN {X 0,Y 495.892,Z 144.214,A -85,B 0,C 180,E1 -6294.306,E2 -6294.306} C_VEL
LIN {X 0,Y 495.99,Z 144.195,A -85,B 0,C 180,E1 -6297.563,E2 -6297.563} C_VEL
LIN {X 0,Y 496.001,Z 144.191,A -85,B 0,C 180,E1 -6300.811,E2 -6300.811} C_VEL
LIN {X 0,Y 495.84,Z 144.215,A -85,B 0,C 180,E1 -6303.25,E2 -6303.25} C_VEL
LIN {X 0,Y 495.875,Z 144.214,A -85,B 0,C 180,E1 -6306.51,E2 -6306.51} C_VEL
LIN {X 0,Y 495.838,Z 144.207,A -85,B 0,C 180,E1 -6308.969,E2 -6308.969} C_VEL
LIN {X 0,Y 495.823,Z 144.219,A -85,B 0,C 180,E1 -6312.034,E2 -6312.034} C_VEL
LIN {X 0,Y 495.819,Z 144.221,A -85,B 0,C 180,E1 -6315.451,E2 -6315.451} C_VEL
LIN {X 0,Y 495.802,Z 144.213,A -85,B 0,C 180,E1 -6318.247,E2 -6318.247} C_VEL
LIN {X 0,Y 495.769,Z 144.221,A -85,B 0,C 180,E1 -6320.756,E2 -6320.756} C_VEL
LIN {X 0,Y 495.748,Z 144.232,A -85,B 0,C 180,E1 -6323.387,E2 -6323.387} C_VEL
LIN {X 0,Y 495.794,Z 144.218,A -85,B 0,C 180,E1 -6326.067,E2 -6326.067} C_VEL
LIN {X 0,Y 495.767,Z 144.222,A -85,B 0,C 180,E1 -6328.815,E2 -6328.815} C_VEL
LIN {X 0,Y 495.754,Z 144.232,A -85,B 0,C 180,E1 -6331.726,E2 -6331.726} C_VEL
LIN {X 0,Y 495.772,Z 144.217,A -85,B 0,C 180,E1 -6334.695,E2 -6334.695} C_VEL
LIN {X 0,Y 495.727,Z 144.237,A -85,B 0,C 180,E1 -6337.561,E2 -6337.561} C_VEL
LIN {X 0,Y 495.762,Z 144.223,A -85,B 0,C 180,E1 -6340.7,E2 -6340.7} C_VEL
LIN {X 0,Y 495.73,Z 144.233,A -85,B 0,C 180,E1 -6343.695,E2 -6343.695} C_VEL
LIN {X 0,Y 495.724,Z 144.224,A -85,B 0,C 180,E1 -6346.305,E2 -6346.305} C_VEL
LIN {X 0,Y 495.762,Z 144.221,A -85,B 0,C 180,E1 -6349.3,E2 -6349.3} C_VEL
LIN {X 0,Y 495.727,Z 144.234,A -85,B 0,C 180,E1 -6352.439,E2 -6352.439} C_VEL
LIN {X 0,Y 495.78,Z 144.218,A -85,B 0,C 180,E1 -6355.457,E2 -6355.457} C_VEL
LIN {X 0,Y 495.755,Z 144.231,A -85,B 0,C 180,E1 -6358.364,E2 -6358.364} C_VEL
LIN {X 0,Y 495.759,Z 144.225,A -85,B 0,C 180,E1 -6360.75,E2 -6360.75} C_VEL
LIN {X 0,Y 495.097,Z 144.311,A -85,B 0,C 180,E1 -6361.429,E2 -6361.429} C_VEL
LIN {X 0,Y 492.236,Z 144.67,A -85,B 0,C 180,E1 -6362.531,E2 -6362.531} C_VEL
LIN {X 0,Y 489.827,Z 144.968,A -85,B 0,C 180,E1 -6363.42,E2 -6363.42} C_VEL
LIN {X 0,Y 488.811,Z 145.096,A -85,B 0,C 180,E1 -6364.106,E2 -6364.106} C_VEL
LIN {X 0,Y 488.738,Z 145.107,A -85,B 0,C 180,E1 -6364.338,E2 -6364.338} C_VEL
LIN {X 0,Y 488.724,Z 145.107,A -85,B 0,C 180,E1 -6367.153,E2 -6367.153} C_VEL
LIN {X 0,Y 488.725,Z 145.106,A -85,B 0,C 180,E1 -6369.811,E2 -6369.811} C_VEL
LIN {X 0,Y 488.731,Z 145.11,A -85,B 0,C 180,E1 -6372.424,E2 -6372.424} C_VEL
LIN {X 0,Y 488.758,Z 145.103,A -85,B 0,C 180,E1 -6375,E2 -6375} C_VEL
LIN {X 0,Y 488.802,Z 145.101,A -85,B 0,C 180,E1 -6378.388,E2 -6378.388} C_VEL
LIN {X 0,Y 488.815,Z 145.098,A -85,B 0,C 180,E1 -6381.734,E2 -6381.734} C_VEL
LIN {X 0,Y 488.853,Z 145.095,A -85,B 0,C 180,E1 -6384.224,E2 -6384.224} C_VEL
LIN {X 0,Y 488.959,Z 145.079,A -85,B 0,C 180,E1 -6387.529,E2 -6387.529} C_VEL
LIN {X 0,Y 488.951,Z 145.078,A -85,B 0,C 180,E1 -6390.824,E2 -6390.824} C_VEL
LIN {X 0,Y 488.959,Z 145.079,A -85,B 0,C 180,E1 -6392.471,E2 -6392.471} C_VEL
LIN {X 0,Y 488.853,Z 145.095,A -85,B 0,C 180,E1 -6395.776,E2 -6395.776} C_VEL
LIN {X 0,Y 488.815,Z 145.098,A -85,B 0,C 180,E1 -6398.266,E2 -6398.266} C_VEL
LIN {X 0,Y 488.802,Z 145.101,A -85,B 0,C 180,E1 -6401.612,E2 -6401.612} C_VEL
LIN {X 0,Y 488.758,Z 145.103,A -85,B 0,C 180,E1 -6405,E2 -6405} C_VEL
LIN {X 0,Y 488.751,Z 145.102,A -85,B 0,C 180,E1 -6408.442,E2 -6408.442} C_VEL
LIN {X 0,Y 488.703,Z 145.112,A -85,B 0,C 180,E1 -6411.071,E2 -6411.071} C_VEL
LIN {X 0,Y 488.69,Z 145.112,A -85,B 0,C 180,E1 -6413.745,E2 -6413.745} C_VEL
LIN {X 0,Y 488.788,Z 145.101,A -85,B 0,C 180,E1 -6416.944,E2 -6416.944} C_VEL
LIN {X 0,Y 488.73,Z 145.1,A -85,B 0,C 180,E1 -6420.218,E2 -6420.218} C_VEL
LIN {X 0,Y 488.731,Z 145.098,A -85,B 0,C 180,E1 -6423.484,E2 -6423.484} C_VEL
LIN {X 0,Y 488.683,Z 145.105,A -85,B 0,C 180,E1 -6426.355,E2 -6426.355} C_VEL
LIN {X 0,Y 488.697,Z 145.107,A -85,B 0,C 180,E1 -6429.254,E2 -6429.254} C_VEL
LIN {X 0,Y 488.703,Z 145.087,A -85,B 0,C 180,E1 -6431.6,E2 -6431.6} C_VEL
LIN {X 0,Y 488.707,Z 145.106,A -85,B 0,C 180,E1 -6434.801,E2 -6434.801} C_VEL
LIN {X 0,Y 488.69,Z 145.107,A -85,B 0,C 180,E1 -6437.475,E2 -6437.475} C_VEL
LIN {X 0,Y 488.727,Z 145.097,A -85,B 0,C 180,E1 -6439.677,E2 -6439.677} C_VEL
LIN {X 0,Y 488.678,Z 145.113,A -85,B 0,C 180,E1 -6442.842,E2 -6442.842} C_VEL
LIN {X 0,Y 488.73,Z 145.095,A -85,B 0,C 180,E1 -6445.888,E2 -6445.888} C_VEL
LIN {X 0,Y 488.689,Z 145.111,A -85,B 0,C 180,E1 -6448.821,E2 -6448.821} C_VEL
LIN {X 0,Y 488.74,Z 145.098,A -85,B 0,C 180,E1 -6451.672,E2 -6451.672} C_VEL
LIN {X 0,Y 488.746,Z 145.104,A -85,B 0,C 180,E1 -6454.445,E2 -6454.445} C_VEL
LIN {X 0,Y 488.723,Z 145.103,A -85,B 0,C 180,E1 -6457.154,E2 -6457.154} C_VEL
LIN {X 0,Y 488.72,Z 145.103,A -85,B 0,C 180,E1 -6459.811,E2 -6459.811} C_VEL
LIN {X 0,Y 488.73,Z 145.103,A -85,B 0,C 180,E1 -6462.424,E2 -6462.424} C_VEL
LIN {X 0,Y 488.757,Z 145.099,A -85,B 0,C 180,E1 -6465,E2 -6465} C_VEL
LIN {X 0,Y 488.801,Z 145.088,A -85,B 0,C 180,E1 -6468.388,E2 -6468.388} C_VEL
LIN {X 0,Y 488.813,Z 145.088,A -85,B 0,C 180,E1 -6471.734,E2 -6471.734} C_VEL
LIN {X 0,Y 488.851,Z 145.09,A -85,B 0,C 180,E1 -6474.225,E2 -6474.225} C_VEL
LIN {X 0,Y 488.957,Z 145.077,A -85,B 0,C 180,E1 -6477.529,E2 -6477.529} C_VEL
LIN {X 0,Y 488.966,Z 145.065,A -85,B 0,C 180,E1 -6480,E2 -6480} C_VEL
LIN {X 0,Y 488.957,Z 145.071,A -85,B 0,C 180,E1 -6482.472,E2 -6482.472} C_VEL
LIN {X 0,Y 488.851,Z 145.09,A -85,B 0,C 180,E1 -6485.776,E2 -6485.776} C_VEL
LIN {X 0,Y 488.814,Z 145.083,A -85,B 0,C 180,E1 -6488.267,E2 -6488.267} C_VEL
LIN {X 0,Y 488.802,Z 145.094,A -85,B 0,C 180,E1 -6491.613,E2 -6491.613} C_VEL
LIN {X 0,Y 488.759,Z 145.103,A -85,B 0,C 180,E1 -6495.001,E2 -6495.001} C_VEL
LIN {X 0,Y 488.753,Z 145.089,A -85,B 0,C 180,E1 -6498.443,E2 -6498.443} C_VEL
LIN {X 0,Y 488.704,Z 145.107,A -85,B 0,C 180,E1 -6501.071,E2 -6501.071} C_VEL
LIN {X 0,Y 488.686,Z 145.107,A -85,B 0,C 180,E1 -6503.746,E2 -6503.746} C_VEL
LIN {X 0,Y 488.79,Z 145.091,A -85,B 0,C 180,E1 -6506.944,E2 -6506.944} C_VEL
LIN {X 0,Y 488.708,Z 145.107,A -85,B 0,C 180,E1 -6510.363,E2 -6510.363} C_VEL
LIN {X 0,Y 488.734,Z 145.096,A -85,B 0,C 180,E1 -6513.485,E2 -6513.485} C_VEL
LIN {X 0,Y 488.681,Z 145.11,A -85,B 0,C 180,E1 -6516.355,E2 -6516.355} C_VEL
LIN {X 0,Y 488.699,Z 145.103,A -85,B 0,C 180,E1 -6519.255,E2 -6519.255} C_VEL
LIN {X 0,Y 488.706,Z 145.105,A -85,B 0,C 180,E1 -6521.6,E2 -6521.6} C_VEL
LIN {X 0,Y 488.701,Z 145.109,A -85,B 0,C 180,E1 -6524.803,E2 -6524.803} C_VEL
LIN {X 0,Y 488.692,Z 145.108,A -85,B 0,C 180,E1 -6527.475,E2 -6527.475} C_VEL
LIN {X 0,Y 488.733,Z 145.095,A -85,B 0,C 180,E1 -6529.677,E2 -6529.677} C_VEL
LIN {X 0,Y 488.68,Z 145.11,A -85,B 0,C 180,E1 -6532.842,E2 -6532.842} C_VEL
LIN {X 0,Y 488.732,Z 145.106,A -85,B 0,C 180,E1 -6535.888,E2 -6535.888} C_VEL
LIN {X 0,Y 488.694,Z 145.111,A -85,B 0,C 180,E1 -6538.821,E2 -6538.821} C_VEL
LIN {X 0,Y 488.745,Z 145.107,A -85,B 0,C 180,E1 -6541.672,E2 -6541.672} C_VEL
LIN {X 0,Y 488.806,Z 145.139,A -85,B 0,C 180,E1 -6543.054,E2 -6543.054} C_VEL
LIN {X 0,Y 490.24,Z 153.51,A -85,B 0,C 180,E1 -6545.046,E2 -6545.046} C_VEL
LIN {X 0,Y 490.005,Z 162.04,A -85,B 0,C 180,E1 -6546.909,E2 -6546.909} C_VEL
LIN {X 0,Y 489.517,Z 176.942,A -85,B 0,C 180,E1 -6550.064,E2 -6550.064} C_VEL
LIN {X 0,Y 489.022,Z 190.361,A -85,B 0,C 180,E1 -6552.866,E2 -6552.866} C_VEL
LIN {X 0,Y 488.955,Z 194.443,A -85,B 0,C 180,E1 -6553.713,E2 -6553.713} C_VEL
LIN {X 0,Y 490.57,Z 204.046,A -85,B 0,C 180,E1 -6553.941,E2 -6553.941} C_VEL
LIN {X 0,Y 491.656,Z 211.943,A -85,B 0,C 180,E1 -6554.094,E2 -6554.094} C_VEL
LIN {X 0,Y 491.171,Z 299.236,A -85,B 0,C 180,E1 -6555.393,E2 -6555.393} C_VEL
LIN {X 0,Y 490.951,Z 309.131,A -85,B 0,C 180,E1 -6555.625,E2 -6555.625} C_VEL
LIN {X 0,Y 490.697,Z 319.108,A -85,B 0,C 180,E1 -6555.961,E2 -6555.961} C_VEL
LIN {X 0,Y 490.32,Z 329.471,A -85,B 0,C 180,E1 -6556.426,E2 -6556.426} C_VEL
LIN {X 0,Y 490.02,Z 338.611,A -85,B 0,C 180,E1 -6556.945,E2 -6556.945} C_VEL
LIN {X 0,Y 489.674,Z 347.607,A -85,B 0,C 180,E1 -6557.568,E2 -6557.568} C_VEL
LIN {X 0,Y 489.344,Z 356.337,A -85,B 0,C 180,E1 -6558.296,E2 -6558.296} C_VEL
LIN {X 0,Y 489.098,Z 363.736,A -85,B 0,C 180,E1 -6559.024,E2 -6559.024} C_VEL
LIN {X 0,Y 488.789,Z 370.956,A -85,B 0,C 180,E1 -6559.855,E2 -6559.855} C_VEL
LIN {X 0,Y 488.539,Z 377.158,A -85,B 0,C 180,E1 -6560.686,E2 -6560.686} C_VEL
LIN {X 0,Y 488.314,Z 383.695,A -85,B 0,C 180,E1 -6561.725,E2 -6561.725} C_VEL
LIN {X 0,Y 488.186,Z 388.196,A -85,B 0,C 180,E1 -6562.556,E2 -6562.556} C_VEL
LIN {X 0,Y 488.016,Z 393.689,A -85,B 0,C 180,E1 -6563.801,E2 -6563.801} C_VEL
LIN {X 0,Y 487.968,Z 398.006,A -85,B 0,C 180,E1 -6565.043,E2 -6565.043} C_VEL
LIN {X 0,Y 487.928,Z 400.369,A -85,B 0,C 180,E1 -6565.87,E2 -6565.87} C_VEL
LIN {X 0,Y 487.965,Z 402.167,A -85,B 0,C 180,E1 -6566.697,E2 -6566.697} C_VEL
LIN {X 0,Y 487.891,Z 404.605,A -85,B 0,C 180,E1 -6568.349,E2 -6568.349} C_VEL
LIN {X 0,Y 487.836,Z 405.191,A -85,B 0,C 180,E1 -6569.175,E2 -6569.175} C_VEL
LIN {X 0,Y 487.836,Z 405.191,A -85,B 0,C 180,E1 -6570.825,E2 -6570.825} C_VEL
LIN {X 0,Y 487.891,Z 404.605,A -85,B 0,C 180,E1 -6571.651,E2 -6571.651} C_VEL
LIN {X 0,Y 487.965,Z 402.167,A -85,B 0,C 180,E1 -6573.303,E2 -6573.303} C_VEL
LIN {X 0,Y 487.922,Z 399.221,A -85,B 0,C 180,E1 -6574.544,E2 -6574.544} C_VEL
LIN {X 0,Y 488.012,Z 395.238,A -85,B 0,C 180,E1 -6575.786,E2 -6575.786} C_VEL
LIN {X 0,Y 488.044,Z 392.025,A -85,B 0,C 180,E1 -6576.615,E2 -6576.615} C_VEL
LIN {X 0,Y 488.221,Z 386.005,A -85,B 0,C 180,E1 -6577.86,E2 -6577.86} C_VEL
LIN {X 0,Y 488.441,Z 379.91,A -85,B 0,C 180,E1 -6578.898,E2 -6578.898} C_VEL
LIN {X 0,Y 488.671,Z 374.21,A -85,B 0,C 180,E1 -6579.729,E2 -6579.729} C_VEL
LIN {X 0,Y 488.984,Z 365.654,A -85,B 0,C 180,E1 -6580.769,E2 -6580.769} C_VEL
LIN {X 0,Y 489.304,Z 357.473,A -85,B 0,C 180,E1 -6581.6,E2 -6581.6} C_VEL
LIN {X 0,Y 489.594,Z 348.958,A -85,B 0,C 180,E1 -6582.329,E2 -6582.329} C_VEL
LIN {X 0,Y 489.964,Z 340.245,A -85,B 0,C 180,E1 -6582.951,E2 -6582.951} C_VEL
LIN {X 0,Y 490.279,Z 330.478,A -85,B 0,C 180,E1 -6583.523,E2 -6583.523} C_VEL
LIN {X 0,Y 490.621,Z 320.395,A -85,B 0,C 180,E1 -6583.988,E2 -6583.988} C_VEL
LIN {X 0,Y 490.877,Z 310.879,A -85,B 0,C 180,E1 -6584.325,E2 -6584.325} C_VEL
LIN {X 0,Y 491.108,Z 300.567,A -85,B 0,C 180,E1 -6584.582,E2 -6584.582} C_VEL
LIN {X 0,Y 491.475,Z 245.034,A -85,B 0,C 180,E1 -6585.42,E2 -6585.42} C_VEL
LIN {X 0,Y 491.554,Z 209.969,A -85,B 0,C 180,E1 -6585.938,E2 -6585.938} C_VEL
LIN {X 0,Y 488.944,Z 194.572,A -85,B 0,C 180,E1 -6586.278,E2 -6586.278} C_VEL
LIN {X 0,Y 488.928,Z 193.753,A -85,B 0,C 180,E1 -6586.385,E2 -6586.385} C_VEL
LIN {X 0,Y 489.312,Z 182.231,A -85,B 0,C 180,E1 -6588.866,E2 -6588.866} C_VEL
LIN {X 0,Y 489.72,Z 169.765,A -85,B 0,C 180,E1 -6591.465,E2 -6591.465} C_VEL
LIN {X 0,Y 490.333,Z 155.267,A -85,B 0,C 180,E1 -6594.561,E2 -6594.561} C_VEL
LIN {X 0,Y 489.553,Z 149.124,A -85,B 0,C 180,E1 -6595.967,E2 -6595.967} C_VEL
LIN {X 0,Y 488.792,Z 145.12,A -85,B 0,C 180,E1 -6596.962,E2 -6596.962} C_VEL
LIN {X 0,Y 488.712,Z 145.112,A -85,B 0,C 180,E1 -6600.362,E2 -6600.362} C_VEL
LIN {X 0,Y 488.736,Z 145.106,A -85,B 0,C 180,E1 -6603.484,E2 -6603.484} C_VEL
LIN {X 0,Y 488.683,Z 145.11,A -85,B 0,C 180,E1 -6606.354,E2 -6606.354} C_VEL
LIN {X 0,Y 488.702,Z 145.108,A -85,B 0,C 180,E1 -6609.254,E2 -6609.254} C_VEL
LIN {X 0,Y 488.707,Z 145.104,A -85,B 0,C 180,E1 -6611.599,E2 -6611.599} C_VEL
LIN {X 0,Y 488.701,Z 145.106,A -85,B 0,C 180,E1 -6614.802,E2 -6614.802} C_VEL
LIN {X 0,Y 488.691,Z 145.116,A -85,B 0,C 180,E1 -6617.474,E2 -6617.474} C_VEL
LIN {X 0,Y 488.732,Z 145.103,A -85,B 0,C 180,E1 -6619.676,E2 -6619.676} C_VEL
LIN {X 0,Y 488.678,Z 145.111,A -85,B 0,C 180,E1 -6622.84,E2 -6622.84} C_VEL
LIN {X 0,Y 488.73,Z 145.097,A -85,B 0,C 180,E1 -6625.887,E2 -6625.887} C_VEL
LIN {X 0,Y 488.691,Z 145.11,A -85,B 0,C 180,E1 -6628.82,E2 -6628.82} C_VEL
LIN {X 0,Y 488.743,Z 145.096,A -85,B 0,C 180,E1 -6631.671,E2 -6631.671} C_VEL
LIN {X 0,Y 488.745,Z 145.095,A -85,B 0,C 180,E1 -6634.444,E2 -6634.444} C_VEL
LIN {X 0,Y 488.72,Z 145.108,A -85,B 0,C 180,E1 -6637.153,E2 -6637.153} C_VEL
LIN {X 0,Y 488.723,Z 145.096,A -85,B 0,C 180,E1 -6639.81,E2 -6639.81} C_VEL
LIN {X 0,Y 488.731,Z 145.094,A -85,B 0,C 180,E1 -6642.423,E2 -6642.423} C_VEL
LIN {X 0,Y 488.759,Z 145.103,A -85,B 0,C 180,E1 -6644.999,E2 -6644.999} C_VEL
LIN {X 0,Y 488.802,Z 145.094,A -85,B 0,C 180,E1 -6648.387,E2 -6648.387} C_VEL
LIN {X 0,Y 488.814,Z 145.083,A -85,B 0,C 180,E1 -6651.733,E2 -6651.733} C_VEL
LIN {X 0,Y 488.851,Z 145.09,A -85,B 0,C 180,E1 -6654.224,E2 -6654.224} C_VEL
LIN {X 0,Y 488.957,Z 145.071,A -85,B 0,C 180,E1 -6657.528,E2 -6657.528} C_VEL
LIN {X 0,Y 488.951,Z 145.068,A -85,B 0,C 180,E1 -6660.823,E2 -6660.823} C_VEL
LIN {X 0,Y 488.957,Z 145.077,A -85,B 0,C 180,E1 -6662.471,E2 -6662.471} C_VEL
LIN {X 0,Y 488.851,Z 145.09,A -85,B 0,C 180,E1 -6665.775,E2 -6665.775} C_VEL
LIN {X 0,Y 488.813,Z 145.088,A -85,B 0,C 180,E1 -6668.266,E2 -6668.266} C_VEL
LIN {X 0,Y 488.801,Z 145.088,A -85,B 0,C 180,E1 -6671.612,E2 -6671.612} C_VEL
LIN {X 0,Y 488.757,Z 145.099,A -85,B 0,C 180,E1 -6675,E2 -6675} C_VEL
LIN {X 0,Y 488.75,Z 145.089,A -85,B 0,C 180,E1 -6678.442,E2 -6678.442} C_VEL
LIN {X 0,Y 488.702,Z 145.102,A -85,B 0,C 180,E1 -6681.07,E2 -6681.07} C_VEL
LIN {X 0,Y 488.69,Z 145.115,A -85,B 0,C 180,E1 -6683.745,E2 -6683.745} C_VEL
LIN {X 0,Y 488.794,Z 145.087,A -85,B 0,C 180,E1 -6686.945,E2 -6686.945} C_VEL
LIN {X 0,Y 488.705,Z 145.106,A -85,B 0,C 180,E1 -6690.363,E2 -6690.363} C_VEL
LIN {X 0,Y 488.731,Z 145.102,A -85,B 0,C 180,E1 -6693.484,E2 -6693.484} C_VEL
LIN {X 0,Y 488.684,Z 145.107,A -85,B 0,C 180,E1 -6696.356,E2 -6696.356} C_VEL
LIN {X 0,Y 488.696,Z 145.112,A -85,B 0,C 180,E1 -6699.254,E2 -6699.254} C_VEL
LIN {X 0,Y 488.719,Z 145.107,A -85,B 0,C 180,E1 -6701.602,E2 -6701.602} C_VEL
LIN {X 0,Y 488.707,Z 145.108,A -85,B 0,C 180,E1 -6704.801,E2 -6704.801} C_VEL
LIN {X 0,Y 488.686,Z 145.091,A -85,B 0,C 180,E1 -6707.474,E2 -6707.474} C_VEL
LIN {X 0,Y 488.728,Z 145.1,A -85,B 0,C 180,E1 -6709.677,E2 -6709.677} C_VEL
LIN {X 0,Y 488.678,Z 145.117,A -85,B 0,C 180,E1 -6712.841,E2 -6712.841} C_VEL
LIN {X 0,Y 488.73,Z 145.094,A -85,B 0,C 180,E1 -6715.888,E2 -6715.888} C_VEL
LIN {X 0,Y 488.714,Z 145.11,A -85,B 0,C 180,E1 -6718.822,E2 -6718.822} C_VEL
LIN {X 0,Y 488.742,Z 145.1,A -85,B 0,C 180,E1 -6721.671,E2 -6721.671} C_VEL
LIN {X 0,Y 488.738,Z 145.107,A -85,B 0,C 180,E1 -6724.338,E2 -6724.338} C_VEL
LIN {X 0,Y 488.094,Z 145.192,A -85,B 0,C 180,E1 -6725.026,E2 -6725.026} C_VEL
LIN {X 0,Y 485.228,Z 145.547,A -85,B 0,C 180,E1 -6726.142,E2 -6726.142} C_VEL
LIN {X 0,Y 482.783,Z 145.848,A -85,B 0,C 180,E1 -6727.042,E2 -6727.042} C_VEL
LIN {X 0,Y 481.724,Z 145.978,A -85,B 0,C 180,E1 -6727.737,E2 -6727.737} C_VEL
LIN {X 0,Y 481.635,Z 145.989,A -85,B 0,C 180,E1 -6727.973,E2 -6727.973} C_VEL
LIN {X 0,Y 481.704,Z 145.985,A -85,B 0,C 180,E1 -6730.393,E2 -6730.393} C_VEL
LIN {X 0,Y 481.687,Z 145.984,A -85,B 0,C 180,E1 -6733.034,E2 -6733.034} C_VEL
LIN {X 0,Y 481.686,Z 145.983,A -85,B 0,C 180,E1 -6735.639,E2 -6735.639} C_VEL
LIN {X 0,Y 481.747,Z 145.98,A -85,B 0,C 180,E1 -6738.215,E2 -6738.215} C_VEL
LIN {X 0,Y 481.76,Z 145.976,A -85,B 0,C 180,E1 -6741.612,E2 -6741.612} C_VEL
LIN {X 0,Y 481.814,Z 145.971,A -85,B 0,C 180,E1 -6744.14,E2 -6744.14} C_VEL
LIN {X 0,Y 481.925,Z 145.955,A -85,B 0,C 180,E1 -6747.493,E2 -6747.493} C_VEL
LIN {X 0,Y 481.902,Z 145.957,A -85,B 0,C 180,E1 -6750.836,E2 -6750.836} C_VEL
LIN {X 0,Y 481.926,Z 145.955,A -85,B 0,C 180,E1 -6752.507,E2 -6752.507} C_VEL
LIN {X 0,Y 481.814,Z 145.971,A -85,B 0,C 180,E1 -6755.86,E2 -6755.86} C_VEL
LIN {X 0,Y 481.76,Z 145.976,A -85,B 0,C 180,E1 -6758.388,E2 -6758.388} C_VEL
LIN {X 0,Y 481.747,Z 145.98,A -85,B 0,C 180,E1 -6761.785,E2 -6761.785} C_VEL
LIN {X 0,Y 481.739,Z 145.98,A -85,B 0,C 180,E1 -6765.224,E2 -6765.224} C_VEL
LIN {X 0,Y 481.709,Z 145.98,A -85,B 0,C 180,E1 -6768.722,E2 -6768.722} C_VEL
LIN {X 0,Y 481.643,Z 145.993,A -85,B 0,C 180,E1 -6771.395,E2 -6771.395} C_VEL
LIN {X 0,Y 481.673,Z 145.984,A -85,B 0,C 180,E1 -6774.113,E2 -6774.113} C_VEL
LIN {X 0,Y 481.743,Z 145.98,A -85,B 0,C 180,E1 -6777.139,E2 -6777.139} C_VEL
LIN {X 0,Y 481.684,Z 145.979,A -85,B 0,C 180,E1 -6779.74,E2 -6779.74} C_VEL
LIN {X 0,Y 481.669,Z 145.986,A -85,B 0,C 180,E1 -6782.674,E2 -6782.674} C_VEL
LIN {X 0,Y 481.636,Z 145.983,A -85,B 0,C 180,E1 -6785.709,E2 -6785.709} C_VEL
LIN {X 0,Y 481.667,Z 145.989,A -85,B 0,C 180,E1 -6788.859,E2 -6788.859} C_VEL
LIN {X 0,Y 481.648,Z 145.964,A -85,B 0,C 180,E1 -6791.913,E2 -6791.913} C_VEL
LIN {X 0,Y 481.654,Z 145.979,A -85,B 0,C 180,E1 -6794.457,E2 -6794.457} C_VEL
LIN {X 0,Y 481.649,Z 145.984,A -85,B 0,C 180,E1 -6797.84,E2 -6797.84} C_VEL
LIN {X 0,Y 481.675,Z 145.984,A -85,B 0,C 180,E1 -6800.651,E2 -6800.651} C_VEL
LIN {X 0,Y 481.626,Z 145.987,A -85,B 0,C 180,E1 -6803.376,E2 -6803.376} C_VEL
LIN {X 0,Y 481.704,Z 145.974,A -85,B 0,C 180,E1 -6806.33,E2 -6806.33} C_VEL
LIN {X 0,Y 481.646,Z 145.985,A -85,B 0,C 180,E1 -6809.417,E2 -6809.417} C_VEL
LIN {X 0,Y 481.697,Z 145.976,A -85,B 0,C 180,E1 -6812.168,E2 -6812.168} C_VEL
LIN {X 0,Y 481.714,Z 145.976,A -85,B 0,C 180,E1 -6814.97,E2 -6814.97} C_VEL
LIN {X 0,Y 481.648,Z 145.987,A -85,B 0,C 180,E1 -6817.705,E2 -6817.705} C_VEL
LIN {X 0,Y 481.701,Z 145.969,A -85,B 0,C 180,E1 -6820.393,E2 -6820.393} C_VEL
LIN {X 0,Y 481.686,Z 145.976,A -85,B 0,C 180,E1 -6823.034,E2 -6823.034} C_VEL
LIN {X 0,Y 481.685,Z 145.984,A -85,B 0,C 180,E1 -6825.639,E2 -6825.639} C_VEL
LIN {X 0,Y 481.746,Z 145.968,A -85,B 0,C 180,E1 -6828.215,E2 -6828.215} C_VEL
LIN {X 0,Y 481.758,Z 145.964,A -85,B 0,C 180,E1 -6831.612,E2 -6831.612} C_VEL
LIN {X 0,Y 481.812,Z 145.968,A -85,B 0,C 180,E1 -6834.14,E2 -6834.14} C_VEL
LIN {X 0,Y 481.924,Z 145.953,A -85,B 0,C 180,E1 -6837.493,E2 -6837.493} C_VEL
LIN {X 0,Y 481.937,Z 145.94,A -85,B 0,C 180,E1 -6840,E2 -6840} C_VEL
LIN {X 0,Y 481.924,Z 145.947,A -85,B 0,C 180,E1 -6842.508,E2 -6842.508} C_VEL
LIN {X 0,Y 481.813,Z 145.965,A -85,B 0,C 180,E1 -6845.861,E2 -6845.861} C_VEL
LIN {X 0,Y 481.759,Z 145.962,A -85,B 0,C 180,E1 -6848.389,E2 -6848.389} C_VEL
LIN {X 0,Y 481.748,Z 145.971,A -85,B 0,C 180,E1 -6851.785,E2 -6851.785} C_VEL
LIN {X 0,Y 481.74,Z 145.978,A -85,B 0,C 180,E1 -6855.225,E2 -6855.225} C_VEL
LIN {X 0,Y 481.71,Z 145.968,A -85,B 0,C 180,E1 -6858.722,E2 -6858.722} C_VEL
LIN {X 0,Y 481.643,Z 145.988,A -85,B 0,C 180,E1 -6861.395,E2 -6861.395} C_VEL
LIN {X 0,Y 481.672,Z 145.981,A -85,B 0,C 180,E1 -6864.114,E2 -6864.114} C_VEL
LIN {X 0,Y 481.745,Z 145.968,A -85,B 0,C 180,E1 -6867.14,E2 -6867.14} C_VEL
LIN {X 0,Y 481.677,Z 145.981,A -85,B 0,C 180,E1 -6869.742,E2 -6869.742} C_VEL
LIN {X 0,Y 481.671,Z 145.985,A -85,B 0,C 180,E1 -6872.675,E2 -6872.675} C_VEL
LIN {X 0,Y 481.636,Z 145.984,A -85,B 0,C 180,E1 -6875.71,E2 -6875.71} C_VEL
LIN {X 0,Y 481.669,Z 145.982,A -85,B 0,C 180,E1 -6878.86,E2 -6878.86} C_VEL
LIN {X 0,Y 481.651,Z 145.985,A -85,B 0,C 180,E1 -6881.913,E2 -6881.913} C_VEL
LIN {X 0,Y 481.654,Z 145.987,A -85,B 0,C 180,E1 -6884.458,E2 -6884.458} C_VEL
LIN {X 0,Y 481.647,Z 145.987,A -85,B 0,C 180,E1 -6887.84,E2 -6887.84} C_VEL
LIN {X 0,Y 481.681,Z 145.981,A -85,B 0,C 180,E1 -6890.652,E2 -6890.652} C_VEL
LIN {X 0,Y 481.628,Z 145.987,A -85,B 0,C 180,E1 -6893.377,E2 -6893.377} C_VEL
LIN {X 0,Y 481.711,Z 145.983,A -85,B 0,C 180,E1 -6896.331,E2 -6896.331} C_VEL
LIN {X 0,Y 481.652,Z 145.99,A -85,B 0,C 180,E1 -6899.418,E2 -6899.418} C_VEL
LIN {X 0,Y 481.715,Z 145.98,A -85,B 0,C 180,E1 -6902.558,E2 -6902.558} C_VEL
LIN {X 0,Y 481.799,Z 146.24,A -85,B 0,C 180,E1 -6902.95,E2 -6902.95} C_VEL
LIN {X 0,Y 483.294,Z 155.131,A -85,B 0,C 180,E1 -6905.057,E2 -6905.057} C_VEL
LIN {X 0,Y 482.923,Z 165.393,A -85,B 0,C 180,E1 -6907.316,E2 -6907.316} C_VEL
LIN {X 0,Y 482.441,Z 178.843,A -85,B 0,C 180,E1 -6910.203,E2 -6910.203} C_VEL
LIN {X 0,Y 482.018,Z 190.178,A -85,B 0,C 180,E1 -6912.609,E2 -6912.609} C_VEL
LIN {X 0,Y 481.933,Z 194.22,A -85,B 0,C 180,E1 -6913.465,E2 -6913.465} C_VEL
LIN {X 0,Y 483.249,Z 201.965,A -85,B 0,C 180,E1 -6913.663,E2 -6913.663} C_VEL
LIN {X 0,Y 484.839,Z 212.943,A -85,B 0,C 180,E1 -6913.883,E2 -6913.883} C_VEL
LIN {X 0,Y 484.299,Z 299.045,A -85,B 0,C 180,E1 -6915.181,E2 -6915.181} C_VEL
LIN {X 0,Y 484.07,Z 308.939,A -85,B 0,C 180,E1 -6915.416,E2 -6915.416} C_VEL
LIN {X 0,Y 483.814,Z 318.917,A -85,B 0,C 180,E1 -6915.757,E2 -6915.757} C_VEL
LIN {X 0,Y 483.425,Z 329.28,A -85,B 0,C 180,E1 -6916.228,E2 -6916.228} C_VEL
LIN {X 0,Y 483.097,Z 338.419,A -85,B 0,C 180,E1 -6916.755,E2 -6916.755} C_VEL
LIN {X 0,Y 482.708,Z 347.414,A -85,B 0,C 180,E1 -6917.385,E2 -6917.385} C_VEL
LIN {X 0,Y 482.362,Z 356.164,A -85,B 0,C 180,E1 -6918.125,E2 -6918.125} C_VEL
LIN {X 0,Y 482.116,Z 363.544,A -85,B 0,C 180,E1 -6918.863,E2 -6918.863} C_VEL
LIN {X 0,Y 481.748,Z 370.763,A -85,B 0,C 180,E1 -6919.706,E2 -6919.706} C_VEL
LIN {X 0,Y 481.487,Z 376.965,A -85,B 0,C 180,E1 -6920.549,E2 -6920.549} C_VEL
LIN {X 0,Y 481.264,Z 383.503,A -85,B 0,C 180,E1 -6921.603,E2 -6921.603} C_VEL
LIN {X 0,Y 481.101,Z 388.003,A -85,B 0,C 180,E1 -6922.445,E2 -6922.445} C_VEL
LIN {X 0,Y 480.917,Z 393.959,A -85,B 0,C 180,E1 -6923.834,E2 -6923.834} C_VEL
LIN {X 0,Y 480.898,Z 397.814,A -85,B 0,C 180,E1 -6924.97,E2 -6924.97} C_VEL
LIN {X 0,Y 480.828,Z 400.177,A -85,B 0,C 180,E1 -6925.809,E2 -6925.809} C_VEL
LIN {X 0,Y 480.888,Z 401.975,A -85,B 0,C 180,E1 -6926.649,E2 -6926.649} C_VEL
LIN {X 0,Y 480.793,Z 404.413,A -85,B 0,C 180,E1 -6928.325,E2 -6928.325} C_VEL
LIN {X 0,Y 480.762,Z 405,A -85,B 0,C 180,E1 -6929.162,E2 -6929.162} C_VEL
LIN {X 0,Y 480.762,Z 405,A -85,B 0,C 180,E1 -6930.838,E2 -6930.838} C_VEL
LIN {X 0,Y 480.793,Z 404.413,A -85,B 0,C 180,E1 -6931.675,E2 -6931.675} C_VEL
LIN {X 0,Y 480.888,Z 401.975,A -85,B 0,C 180,E1 -6933.351,E2 -6933.351} C_VEL
LIN {X 0,Y 480.84,Z 399.029,A -85,B 0,C 180,E1 -6934.611,E2 -6934.611} C_VEL
LIN {X 0,Y 480.917,Z 395.045,A -85,B 0,C 180,E1 -6935.871,E2 -6935.871} C_VEL
LIN {X 0,Y 481.02,Z 389.918,A -85,B 0,C 180,E1 -6937.134,E2 -6937.134} C_VEL
LIN {X 0,Y 481.221,Z 384.658,A -85,B 0,C 180,E1 -6938.186,E2 -6938.186} C_VEL
LIN {X 0,Y 481.441,Z 378.341,A -85,B 0,C 180,E1 -6939.24,E2 -6939.24} C_VEL
LIN {X 0,Y 481.673,Z 372.389,A -85,B 0,C 180,E1 -6940.084,E2 -6940.084} C_VEL
LIN {X 0,Y 481.988,Z 365.462,A -85,B 0,C 180,E1 -6940.927,E2 -6940.927} C_VEL
LIN {X 0,Y 482.333,Z 357.281,A -85,B 0,C 180,E1 -6941.77,E2 -6941.77} C_VEL
LIN {X 0,Y 482.637,Z 348.657,A -85,B 0,C 180,E1 -6942.518,E2 -6942.518} C_VEL
LIN {X 0,Y 483.015,Z 340.053,A -85,B 0,C 180,E1 -6943.141,E2 -6943.141} C_VEL
LIN {X 0,Y 483.371,Z 330.286,A -85,B 0,C 180,E1 -6943.72,E2 -6943.72} C_VEL
LIN {X 0,Y 483.709,Z 321.492,A -85,B 0,C 180,E1 -6944.139,E2 -6944.139} C_VEL
LIN {X 0,Y 483.974,Z 311.562,A -85,B 0,C 180,E1 -6944.507,E2 -6944.507} C_VEL
LIN {X 0,Y 484.222,Z 301.707,A -85,B 0,C 180,E1 -6944.768,E2 -6944.768} C_VEL
LIN {X 0,Y 484.479,Z 277.358,A -85,B 0,C 180,E1 -6945.159,E2 -6945.159} C_VEL
LIN {X 0,Y 484.712,Z 210.637,A -85,B 0,C 180,E1 -6946.156,E2 -6946.156} C_VEL
LIN {X 0,Y 481.932,Z 194.429,A -85,B 0,C 180,E1 -6946.519,E2 -6946.519} C_VEL
LIN {X 0,Y 481.916,Z 193.563,A -85,B 0,C 180,E1 -6946.631,E2 -6946.631} C_VEL
LIN {X 0,Y 482.398,Z 181.102,A -85,B 0,C 180,E1 -6949.356,E2 -6949.356} C_VEL
LIN {X 0,Y 482.967,Z 165.443,A -85,B 0,C 180,E1 -6952.682,E2 -6952.682} C_VEL
LIN {X 0,Y 483.325,Z 155.131,A -85,B 0,C 180,E1 -6954.941,E2 -6954.941} C_VEL
LIN {X 0,Y 481.75,Z 146.011,A -85,B 0,C 180,E1 -6957.139,E2 -6957.139} C_VEL
LIN {X 0,Y 481.68,Z 145.983,A -85,B 0,C 180,E1 -6959.741,E2 -6959.741} C_VEL
LIN {X 0,Y 481.673,Z 145.983,A -85,B 0,C 180,E1 -6962.674,E2 -6962.674} C_VEL
LIN {X 0,Y 481.638,Z 145.985,A -85,B 0,C 180,E1 -6965.709,E2 -6965.709} C_VEL
LIN {X 0,Y 481.672,Z 145.981,A -85,B 0,C 180,E1 -6968.858,E2 -6968.858} C_VEL
LIN {X 0,Y 481.652,Z 145.989,A -85,B 0,C 180,E1 -6971.912,E2 -6971.912} C_VEL
LIN {X 0,Y 481.654,Z 145.983,A -85,B 0,C 180,E1 -6974.457,E2 -6974.457} C_VEL
LIN {X 0,Y 481.647,Z 145.988,A -85,B 0,C 180,E1 -6977.839,E2 -6977.839} C_VEL
LIN {X 0,Y 481.66,Z 145.979,A -85,B 0,C 180,E1 -6980.653,E2 -6980.653} C_VEL
LIN {X 0,Y 481.626,Z 145.993,A -85,B 0,C 180,E1 -6983.376,E2 -6983.376} C_VEL
LIN {X 0,Y 481.709,Z 145.97,A -85,B 0,C 180,E1 -6986.329,E2 -6986.329} C_VEL
LIN {X 0,Y 481.649,Z 145.989,A -85,B 0,C 180,E1 -6989.417,E2 -6989.417} C_VEL
LIN {X 0,Y 481.698,Z 145.972,A -85,B 0,C 180,E1 -6992.167,E2 -6992.167} C_VEL
LIN {X 0,Y 481.715,Z 145.977,A -85,B 0,C 180,E1 -6994.969,E2 -6994.969} C_VEL
LIN {X 0,Y 481.646,Z 145.984,A -85,B 0,C 180,E1 -6997.704,E2 -6997.704} C_VEL
LIN {X 0,Y 481.703,Z 145.972,A -85,B 0,C 180,E1 -7000.393,E2 -7000.393} C_VEL
LIN {X 0,Y 481.688,Z 145.98,A -85,B 0,C 180,E1 -7003.033,E2 -7003.033} C_VEL
LIN {X 0,Y 481.687,Z 145.979,A -85,B 0,C 180,E1 -7005.638,E2 -7005.638} C_VEL
LIN {X 0,Y 481.748,Z 145.971,A -85,B 0,C 180,E1 -7008.215,E2 -7008.215} C_VEL
LIN {X 0,Y 481.759,Z 145.962,A -85,B 0,C 180,E1 -7011.611,E2 -7011.611} C_VEL
LIN {X 0,Y 481.813,Z 145.965,A -85,B 0,C 180,E1 -7014.139,E2 -7014.139} C_VEL
LIN {X 0,Y 481.924,Z 145.947,A -85,B 0,C 180,E1 -7017.492,E2 -7017.492} C_VEL
LIN {X 0,Y 481.902,Z 145.946,A -85,B 0,C 180,E1 -7020.835,E2 -7020.835} C_VEL
LIN {X 0,Y 481.924,Z 145.953,A -85,B 0,C 180,E1 -7022.507,E2 -7022.507} C_VEL
LIN {X 0,Y 481.812,Z 145.968,A -85,B 0,C 180,E1 -7025.86,E2 -7025.86} C_VEL
LIN {X 0,Y 481.758,Z 145.964,A -85,B 0,C 180,E1 -7028.388,E2 -7028.388} C_VEL
LIN {X 0,Y 481.746,Z 145.968,A -85,B 0,C 180,E1 -7031.785,E2 -7031.785} C_VEL
LIN {X 0,Y 481.738,Z 145.974,A -85,B 0,C 180,E1 -7035.224,E2 -7035.224} C_VEL
LIN {X 0,Y 481.707,Z 145.964,A -85,B 0,C 180,E1 -7038.721,E2 -7038.721} C_VEL
LIN {X 0,Y 481.642,Z 145.984,A -85,B 0,C 180,E1 -7041.394,E2 -7041.394} C_VEL
LIN {X 0,Y 481.673,Z 145.984,A -85,B 0,C 180,E1 -7044.113,E2 -7044.113} C_VEL
LIN {X 0,Y 481.747,Z 145.966,A -85,B 0,C 180,E1 -7047.14,E2 -7047.14} C_VEL
LIN {X 0,Y 481.674,Z 145.988,A -85,B 0,C 180,E1 -7049.741,E2 -7049.741} C_VEL
LIN {X 0,Y 481.668,Z 145.981,A -85,B 0,C 180,E1 -7052.674,E2 -7052.674} C_VEL
LIN {X 0,Y 481.638,Z 145.99,A -85,B 0,C 180,E1 -7055.709,E2 -7055.709} C_VEL
LIN {X 0,Y 481.666,Z 145.985,A -85,B 0,C 180,E1 -7058.859,E2 -7058.859} C_VEL
LIN {X 0,Y 481.657,Z 145.984,A -85,B 0,C 180,E1 -7061.914,E2 -7061.914} C_VEL
LIN {X 0,Y 481.655,Z 145.984,A -85,B 0,C 180,E1 -7064.457,E2 -7064.457} C_VEL
LIN {X 0,Y 481.642,Z 145.965,A -85,B 0,C 180,E1 -7067.839,E2 -7067.839} C_VEL
LIN {X 0,Y 481.676,Z 145.98,A -85,B 0,C 180,E1 -7070.651,E2 -7070.651} C_VEL
LIN {X 0,Y 481.627,Z 145.986,A -85,B 0,C 180,E1 -7073.375,E2 -7073.375} C_VEL
LIN {X 0,Y 481.705,Z 145.971,A -85,B 0,C 180,E1 -7076.33,E2 -7076.33} C_VEL
LIN {X 0,Y 481.66,Z 145.982,A -85,B 0,C 180,E1 -7079.415,E2 -7079.415} C_VEL
LIN {X 0,Y 481.697,Z 145.979,A -85,B 0,C 180,E1 -7082.168,E2 -7082.168} C_VEL
LIN {X 0,Y 481.714,Z 145.982,A -85,B 0,C 180,E1 -7084.97,E2 -7084.97} C_VEL
LIN {X 0,Y 481.635,Z 145.989,A -85,B 0,C 180,E1 -7087.973,E2 -7087.973} C_VEL
LIN {X 0,Y 480.966,Z 146.077,A -85,B 0,C 180,E1 -7088.671,E2 -7088.671} C_VEL
LIN {X 0,Y 478.138,Z 146.425,A -85,B 0,C 180,E1 -7089.805,E2 -7089.805} C_VEL
LIN {X 0,Y 475.754,Z 146.726,A -85,B 0,C 180,E1 -7090.72,E2 -7090.72} C_VEL
LIN {X 0,Y 474.734,Z 146.849,A -85,B 0,C 180,E1 -7091.425,E2 -7091.425} C_VEL
LIN {X 0,Y 474.652,Z 146.859,A -85,B 0,C 180,E1 -7091.664,E2 -7091.664} C_VEL
LIN {X 0,Y 474.696,Z 146.858,A -85,B 0,C 180,E1 -7094.544,E2 -7094.544} C_VEL
LIN {X 0,Y 474.701,Z 146.857,A -85,B 0,C 180,E1 -7098.038,E2 -7098.038} C_VEL
LIN {X 0,Y 474.725,Z 146.851,A -85,B 0,C 180,E1 -7101.487,E2 -7101.487} C_VEL
LIN {X 0,Y 474.776,Z 146.848,A -85,B 0,C 180,E1 -7104.052,E2 -7104.052} C_VEL
LIN {X 0,Y 474.891,Z 146.831,A -85,B 0,C 180,E1 -7107.455,E2 -7107.455} C_VEL
LIN {X 0,Y 474.909,Z 146.832,A -85,B 0,C 180,E1 -7110,E2 -7110} C_VEL
LIN {X 0,Y 474.892,Z 146.831,A -85,B 0,C 180,E1 -7112.545,E2 -7112.545} C_VEL
LIN {X 0,Y 474.776,Z 146.848,A -85,B 0,C 180,E1 -7115.948,E2 -7115.948} C_VEL
LIN {X 0,Y 474.725,Z 146.851,A -85,B 0,C 180,E1 -7118.513,E2 -7118.513} C_VEL
LIN {X 0,Y 474.701,Z 146.857,A -85,B 0,C 180,E1 -7121.962,E2 -7121.962} C_VEL
LIN {X 0,Y 474.696,Z 146.858,A -85,B 0,C 180,E1 -7125.456,E2 -7125.456} C_VEL
LIN {X 0,Y 474.662,Z 146.86,A -85,B 0,C 180,E1 -7129.01,E2 -7129.01} C_VEL
LIN {X 0,Y 474.587,Z 146.871,A -85,B 0,C 180,E1 -7131.729,E2 -7131.729} C_VEL
LIN {X 0,Y 474.655,Z 146.858,A -85,B 0,C 180,E1 -7134.493,E2 -7134.493} C_VEL
LIN {X 0,Y 474.695,Z 146.857,A -85,B 0,C 180,E1 -7137.339,E2 -7137.339} C_VEL
LIN {X 0,Y 474.613,Z 146.861,A -85,B 0,C 180,E1 -7140.813,E2 -7140.813} C_VEL
LIN {X 0,Y 474.633,Z 146.85,A -85,B 0,C 180,E1 -7143.984,E2 -7143.984} C_VEL
LIN {X 0,Y 474.569,Z 146.869,A -85,B 0,C 180,E1 -7146.9,E2 -7146.9} C_VEL
LIN {X 0,Y 474.623,Z 146.856,A -85,B 0,C 180,E1 -7149.648,E2 -7149.648} C_VEL
LIN {X 0,Y 474.61,Z 146.847,A -85,B 0,C 180,E1 -7152.934,E2 -7152.934} C_VEL
LIN {X 0,Y 474.61,Z 146.861,A -85,B 0,C 180,E1 -7155.896,E2 -7155.896} C_VEL
LIN {X 0,Y 474.627,Z 146.857,A -85,B 0,C 180,E1 -7159.04,E2 -7159.04} C_VEL
LIN {X 0,Y 474.605,Z 146.863,A -85,B 0,C 180,E1 -7161.704,E2 -7161.704} C_VEL
LIN {X 0,Y 474.625,Z 146.856,A -85,B 0,C 180,E1 -7164.726,E2 -7164.726} C_VEL
LIN {X 0,Y 474.632,Z 146.858,A -85,B 0,C 180,E1 -7167.788,E2 -7167.788} C_VEL
LIN {X 0,Y 474.619,Z 146.858,A -85,B 0,C 180,E1 -7170.885,E2 -7170.885} C_VEL
LIN {X 0,Y 474.661,Z 146.847,A -85,B 0,C 180,E1 -7173.629,E2 -7173.629} C_VEL
LIN {X 0,Y 474.631,Z 146.862,A -85,B 0,C 180,E1 -7176.641,E2 -7176.641} C_VEL
LIN {X 0,Y 474.65,Z 146.85,A -85,B 0,C 180,E1 -7180.09,E2 -7180.09} C_VEL
LIN {X 0,Y 474.646,Z 146.854,A -85,B 0,C 180,E1 -7182.775,E2 -7182.775} C_VEL
LIN {X 0,Y 474.644,Z 146.859,A -85,B 0,C 180,E1 -7185.421,E2 -7185.421} C_VEL
LIN {X 0,Y 474.699,Z 146.848,A -85,B 0,C 180,E1 -7188.038,E2 -7188.038} C_VEL
LIN {X 0,Y 474.724,Z 146.839,A -85,B 0,C 180,E1 -7191.487,E2 -7191.487} C_VEL
LIN {X 0,Y 474.775,Z 146.845,A -85,B 0,C 180,E1 -7194.053,E2 -7194.053} C_VEL
LIN {X 0,Y 474.89,Z 146.829,A -85,B 0,C 180,E1 -7197.456,E2 -7197.456} C_VEL
LIN {X 0,Y 474.908,Z 146.814,A -85,B 0,C 180,E1 -7200,E2 -7200} C_VEL
LIN {X 0,Y 474.89,Z 146.823,A -85,B 0,C 180,E1 -7202.545,E2 -7202.545} C_VEL
LIN {X 0,Y 474.775,Z 146.841,A -85,B 0,C 180,E1 -7205.948,E2 -7205.948} C_VEL
LIN {X 0,Y 474.724,Z 146.838,A -85,B 0,C 180,E1 -7208.514,E2 -7208.514} C_VEL
LIN {X 0,Y 474.701,Z 146.847,A -85,B 0,C 180,E1 -7211.963,E2 -7211.963} C_VEL
LIN {X 0,Y 474.697,Z 146.852,A -85,B 0,C 180,E1 -7215.456,E2 -7215.456} C_VEL
LIN {X 0,Y 474.662,Z 146.846,A -85,B 0,C 180,E1 -7219.011,E2 -7219.011} C_VEL
LIN {X 0,Y 474.586,Z 146.864,A -85,B 0,C 180,E1 -7221.729,E2 -7221.729} C_VEL
LIN {X 0,Y 474.655,Z 146.857,A -85,B 0,C 180,E1 -7224.494,E2 -7224.494} C_VEL
LIN {X 0,Y 474.679,Z 146.848,A -85,B 0,C 180,E1 -7227.335,E2 -7227.335} C_VEL
LIN {X 0,Y 474.604,Z 146.863,A -85,B 0,C 180,E1 -7230.231,E2 -7230.231} C_VEL
LIN {X 0,Y 474.642,Z 146.852,A -85,B 0,C 180,E1 -7233.221,E2 -7233.221} C_VEL
LIN {X 0,Y 474.588,Z 146.865,A -85,B 0,C 180,E1 -7236.324,E2 -7236.324} C_VEL
LIN {X 0,Y 474.617,Z 146.856,A -85,B 0,C 180,E1 -7239.647,E2 -7239.647} C_VEL
LIN {X 0,Y 474.623,Z 146.864,A -85,B 0,C 180,E1 -7242.237,E2 -7242.237} C_VEL
LIN {X 0,Y 474.616,Z 146.86,A -85,B 0,C 180,E1 -7245.298,E2 -7245.298} C_VEL
LIN {X 0,Y 474.62,Z 146.862,A -85,B 0,C 180,E1 -7248.215,E2 -7248.215} C_VEL
LIN {X 0,Y 474.645,Z 146.853,A -85,B 0,C 180,E1 -7250.455,E2 -7250.455} C_VEL
LIN {X 0,Y 474.59,Z 146.866,A -85,B 0,C 180,E1 -7253.677,E2 -7253.677} C_VEL
LIN {X 0,Y 474.644,Z 146.859,A -85,B 0,C 180,E1 -7256.78,E2 -7256.78} C_VEL
LIN {X 0,Y 474.607,Z 146.867,A -85,B 0,C 180,E1 -7259.77,E2 -7259.77} C_VEL
LIN {X 0,Y 474.717,Z 147.034,A -85,B 0,C 180,E1 -7262.716,E2 -7262.716} C_VEL
LIN {X 0,Y 476.28,Z 156.016,A -85,B 0,C 180,E1 -7264.898,E2 -7264.898} C_VEL
LIN {X 0,Y 476.126,Z 163.154,A -85,B 0,C 180,E1 -7266.513,E2 -7266.513} C_VEL
LIN {X 0,Y 475.554,Z 177.646,A -85,B 0,C 180,E1 -7269.678,E2 -7269.678} C_VEL
LIN {X 0,Y 475.051,Z 189.994,A -85,B 0,C 180,E1 -7272.345,E2 -7272.345} C_VEL
LIN {X 0,Y 474.933,Z 193.949,A -85,B 0,C 180,E1 -7273.204,E2 -7273.204} C_VEL
LIN {X 0,Y 475.606,Z 198.051,A -85,B 0,C 180,E1 -7273.335,E2 -7273.335} C_VEL
LIN {X 0,Y 478.033,Z 213.532,A -85,B 0,C 180,E1 -7273.659,E2 -7273.659} C_VEL
LIN {X 0,Y 477.428,Z 298.853,A -85,B 0,C 180,E1 -7274.963,E2 -7274.963} C_VEL
LIN {X 0,Y 477.207,Z 308.748,A -85,B 0,C 180,E1 -7275.201,E2 -7275.201} C_VEL
LIN {X 0,Y 476.944,Z 318.725,A -85,B 0,C 180,E1 -7275.547,E2 -7275.547} C_VEL
LIN {X 0,Y 476.561,Z 328.08,A -85,B 0,C 180,E1 -7275.971,E2 -7275.971} C_VEL
LIN {X 0,Y 476.165,Z 338.227,A -85,B 0,C 180,E1 -7276.558,E2 -7276.558} C_VEL
LIN {X 0,Y 475.746,Z 347.221,A -85,B 0,C 180,E1 -7277.198,E2 -7277.198} C_VEL
LIN {X 0,Y 475.383,Z 356.064,A -85,B 0,C 180,E1 -7277.957,E2 -7277.957} C_VEL
LIN {X 0,Y 475.118,Z 363.351,A -85,B 0,C 180,E1 -7278.697,E2 -7278.697} C_VEL
LIN {X 0,Y 474.737,Z 370.57,A -85,B 0,C 180,E1 -7279.552,E2 -7279.552} C_VEL
LIN {X 0,Y 474.461,Z 376.772,A -85,B 0,C 180,E1 -7280.407,E2 -7280.407} C_VEL
LIN {X 0,Y 474.198,Z 383.31,A -85,B 0,C 180,E1 -7281.477,E2 -7281.477} C_VEL
LIN {X 0,Y 474.03,Z 387.811,A -85,B 0,C 180,E1 -7282.332,E2 -7282.332} C_VEL
LIN {X 0,Y 473.867,Z 393.11,A -85,B 0,C 180,E1 -7283.561,E2 -7283.561} C_VEL
LIN {X 0,Y 473.827,Z 397.623,A -85,B 0,C 180,E1 -7284.894,E2 -7284.894} C_VEL
LIN {X 0,Y 473.735,Z 399.985,A -85,B 0,C 180,E1 -7285.746,E2 -7285.746} C_VEL
LIN {X 0,Y 473.796,Z 401.784,A -85,B 0,C 180,E1 -7286.598,E2 -7286.598} C_VEL
LIN {X 0,Y 473.698,Z 404.222,A -85,B 0,C 180,E1 -7288.3,E2 -7288.3} C_VEL
LIN {X 0,Y 473.69,Z 404.809,A -85,B 0,C 180,E1 -7289.15,E2 -7289.15} C_VEL
LIN {X 0,Y 473.69,Z 404.809,A -85,B 0,C 180,E1 -7290.85,E2 -7290.85} C_VEL
LIN {X 0,Y 473.698,Z 404.222,A -85,B 0,C 180,E1 -7291.7,E2 -7291.7} C_VEL
LIN {X 0,Y 473.796,Z 401.784,A -85,B 0,C 180,E1 -7293.402,E2 -7293.402} C_VEL
LIN {X 0,Y 473.763,Z 398.837,A -85,B 0,C 180,E1 -7294.68,E2 -7294.68} C_VEL
LIN {X 0,Y 473.825,Z 394.853,A -85,B 0,C 180,E1 -7295.96,E2 -7295.96} C_VEL
LIN {X 0,Y 473.947,Z 389.725,A -85,B 0,C 180,E1 -7297.241,E2 -7297.241} C_VEL
LIN {X 0,Y 474.158,Z 384.465,A -85,B 0,C 180,E1 -7298.309,E2 -7298.309} C_VEL
LIN {X 0,Y 474.39,Z 378.148,A -85,B 0,C 180,E1 -7299.379,E2 -7299.379} C_VEL
LIN {X 0,Y 474.638,Z 372.197,A -85,B 0,C 180,E1 -7300.235,E2 -7300.235} C_VEL
LIN {X 0,Y 474.99,Z 365.27,A -85,B 0,C 180,E1 -7301.09,E2 -7301.09} C_VEL
LIN {X 0,Y 475.373,Z 357.089,A -85,B 0,C 180,E1 -7301.945,E2 -7301.945} C_VEL
LIN {X 0,Y 475.693,Z 348.465,A -85,B 0,C 180,E1 -7302.704,E2 -7302.704} C_VEL
LIN {X 0,Y 476.094,Z 339.861,A -85,B 0,C 180,E1 -7303.335,E2 -7303.335} C_VEL
LIN {X 0,Y 476.476,Z 330.095,A -85,B 0,C 180,E1 -7303.922,E2 -7303.922} C_VEL
LIN {X 0,Y 476.818,Z 321.3,A -85,B 0,C 180,E1 -7304.348,E2 -7304.348} C_VEL
LIN {X 0,Y 477.102,Z 311.37,A -85,B 0,C 180,E1 -7304.72,E2 -7304.72} C_VEL
LIN {X 0,Y 477.356,Z 301.516,A -85,B 0,C 180,E1 -7304.985,E2 -7304.985} C_VEL
LIN {X 0,Y 477.64,Z 277.267,A -85,B 0,C 180,E1 -7305.38,E2 -7305.38} C_VEL
LIN {X 0,Y 477.845,Z 211.299,A -85,B 0,C 180,E1 -7306.382,E2 -7306.382} C_VEL
LIN {X 0,Y 474.931,Z 194.38,A -85,B 0,C 180,E1 -7306.761,E2 -7306.761} C_VEL
LIN {X 0,Y 474.922,Z 193.228,A -85,B 0,C 180,E1 -7306.916,E2 -7306.916} C_VEL
LIN {X 0,Y 475.424,Z 180.941,A -85,B 0,C 180,E1 -7309.652,E2 -7309.652} C_VEL
LIN {X 0,Y 476.016,Z 166.357,A -85,B 0,C 180,E1 -7312.803,E2 -7312.803} C_VEL
LIN {X 0,Y 476.4,Z 157.039,A -85,B 0,C 180,E1 -7314.862,E2 -7314.862} C_VEL
LIN {X 0,Y 475.081,Z 148.855,A -85,B 0,C 180,E1 -7316.82,E2 -7316.82} C_VEL
LIN {X 0,Y 474.699,Z 146.876,A -85,B 0,C 180,E1 -7317.368,E2 -7317.368} C_VEL
LIN {X 0,Y 474.606,Z 146.867,A -85,B 0,C 180,E1 -7320.81,E2 -7320.81} C_VEL
LIN {X 0,Y 474.639,Z 146.864,A -85,B 0,C 180,E1 -7323.983,E2 -7323.983} C_VEL
LIN {X 0,Y 474.573,Z 146.866,A -85,B 0,C 180,E1 -7326.899,E2 -7326.899} C_VEL
LIN {X 0,Y 474.628,Z 146.854,A -85,B 0,C 180,E1 -7329.647,E2 -7329.647} C_VEL
LIN {X 0,Y 474.614,Z 146.862,A -85,B 0,C 180,E1 -7332.934,E2 -7332.934} C_VEL
LIN {X 0,Y 474.604,Z 146.866,A -85,B 0,C 180,E1 -7335.894,E2 -7335.894} C_VEL
LIN {X 0,Y 474.627,Z 146.862,A -85,B 0,C 180,E1 -7339.04,E2 -7339.04} C_VEL
LIN {X 0,Y 474.609,Z 146.866,A -85,B 0,C 180,E1 -7341.704,E2 -7341.704} C_VEL
LIN {X 0,Y 474.624,Z 146.859,A -85,B 0,C 180,E1 -7344.725,E2 -7344.725} C_VEL
LIN {X 0,Y 474.635,Z 146.859,A -85,B 0,C 180,E1 -7347.787,E2 -7347.787} C_VEL
LIN {X 0,Y 474.623,Z 146.864,A -85,B 0,C 180,E1 -7350.884,E2 -7350.884} C_VEL
LIN {X 0,Y 474.658,Z 146.85,A -85,B 0,C 180,E1 -7353.628,E2 -7353.628} C_VEL
LIN {X 0,Y 474.633,Z 146.861,A -85,B 0,C 180,E1 -7356.641,E2 -7356.641} C_VEL
LIN {X 0,Y 474.652,Z 146.849,A -85,B 0,C 180,E1 -7360.089,E2 -7360.089} C_VEL
LIN {X 0,Y 474.648,Z 146.852,A -85,B 0,C 180,E1 -7362.774,E2 -7362.774} C_VEL
LIN {X 0,Y 474.645,Z 146.857,A -85,B 0,C 180,E1 -7365.42,E2 -7365.42} C_VEL
LIN {X 0,Y 474.701,Z 146.847,A -85,B 0,C 180,E1 -7368.037,E2 -7368.037} C_VEL
LIN {X 0,Y 474.724,Z 146.838,A -85,B 0,C 180,E1 -7371.486,E2 -7371.486} C_VEL
LIN {X 0,Y 474.775,Z 146.841,A -85,B 0,C 180,E1 -7374.052,E2 -7374.052} C_VEL
LIN {X 0,Y 474.89,Z 146.823,A -85,B 0,C 180,E1 -7377.455,E2 -7377.455} C_VEL
LIN {X 0,Y 474.908,Z 146.814,A -85,B 0,C 180,E1 -7380,E2 -7380} C_VEL
LIN {X 0,Y 474.89,Z 146.829,A -85,B 0,C 180,E1 -7382.544,E2 -7382.544} C_VEL
LIN {X 0,Y 474.775,Z 146.845,A -85,B 0,C 180,E1 -7385.947,E2 -7385.947} C_VEL
LIN {X 0,Y 474.724,Z 146.839,A -85,B 0,C 180,E1 -7388.513,E2 -7388.513} C_VEL
LIN {X 0,Y 474.699,Z 146.848,A -85,B 0,C 180,E1 -7391.962,E2 -7391.962} C_VEL
LIN {X 0,Y 474.695,Z 146.853,A -85,B 0,C 180,E1 -7395.455,E2 -7395.455} C_VEL
LIN {X 0,Y 474.66,Z 146.841,A -85,B 0,C 180,E1 -7399.01,E2 -7399.01} C_VEL
LIN {X 0,Y 474.586,Z 146.867,A -85,B 0,C 180,E1 -7401.728,E2 -7401.728} C_VEL
LIN {X 0,Y 474.655,Z 146.855,A -85,B 0,C 180,E1 -7404.493,E2 -7404.493} C_VEL
LIN {X 0,Y 474.694,Z 146.845,A -85,B 0,C 180,E1 -7407.338,E2 -7407.338} C_VEL
LIN {X 0,Y 474.6,Z 146.864,A -85,B 0,C 180,E1 -7410.81,E2 -7410.81} C_VEL
LIN {X 0,Y 474.633,Z 146.851,A -85,B 0,C 180,E1 -7413.984,E2 -7413.984} C_VEL
LIN {X 0,Y 474.57,Z 146.868,A -85,B 0,C 180,E1 -7416.9,E2 -7416.9} C_VEL
LIN {X 0,Y 474.622,Z 146.858,A -85,B 0,C 180,E1 -7419.647,E2 -7419.647} C_VEL
LIN {X 0,Y 474.63,Z 146.862,A -85,B 0,C 180,E1 -7422.932,E2 -7422.932} C_VEL
LIN {X 0,Y 474.608,Z 146.854,A -85,B 0,C 180,E1 -7425.896,E2 -7425.896} C_VEL
LIN {X 0,Y 474.622,Z 146.846,A -85,B 0,C 180,E1 -7429.041,E2 -7429.041} C_VEL
LIN {X 0,Y 474.606,Z 146.864,A -85,B 0,C 180,E1 -7431.704,E2 -7431.704} C_VEL
LIN {X 0,Y 474.625,Z 146.854,A -85,B 0,C 180,E1 -7434.726,E2 -7434.726} C_VEL
LIN {X 0,Y 474.633,Z 146.86,A -85,B 0,C 180,E1 -7437.788,E2 -7437.788} C_VEL
LIN {X 0,Y 474.627,Z 146.856,A -85,B 0,C 180,E1 -7440.883,E2 -7440.883} C_VEL
LIN {X 0,Y 474.656,Z 146.858,A -85,B 0,C 180,E1 -7443.628,E2 -7443.628} C_VEL
LIN {X 0,Y 474.632,Z 146.867,A -85,B 0,C 180,E1 -7446.641,E2 -7446.641} C_VEL
LIN {X 0,Y 474.653,Z 146.861,A -85,B 0,C 180,E1 -7450.09,E2 -7450.09} C_VEL
LIN {X 0,Y 474.652,Z 146.859,A -85,B 0,C 180,E1 -7451.664,E2 -7451.664} C_VEL
LIN {X 0,Y 473.989,Z 146.947,A -85,B 0,C 180,E1 -7452.373,E2 -7452.373} C_VEL
LIN {X 0,Y 471.138,Z 147.3,A -85,B 0,C 180,E1 -7453.525,E2 -7453.525} C_VEL
LIN {X 0,Y 468.722,Z 147.603,A -85,B 0,C 180,E1 -7454.453,E2 -7454.453} C_VEL
LIN {X 0,Y 467.681,Z 147.728,A -85,B 0,C 180,E1 -7455.17,E2 -7455.17} C_VEL
LIN {X 0,Y 467.593,Z 147.739,A -85,B 0,C 180,E1 -7455.413,E2 -7455.413} C_VEL
LIN {X 0,Y 467.65,Z 147.735,A -85,B 0,C 180,E1 -7458.734,E2 -7458.734} C_VEL
LIN {X 0,Y 467.745,Z 147.724,A -85,B 0,C 180,E1 -7462.228,E2 -7462.228} C_VEL
LIN {X 0,Y 467.722,Z 147.724,A -85,B 0,C 180,E1 -7464.827,E2 -7464.827} C_VEL
LIN {X 0,Y 467.857,Z 147.707,A -85,B 0,C 180,E1 -7467.417,E2 -7467.417} C_VEL
LIN {X 0,Y 467.88,Z 147.708,A -85,B 0,C 180,E1 -7470,E2 -7470} C_VEL
LIN {X 0,Y 467.857,Z 147.707,A -85,B 0,C 180,E1 -7472.583,E2 -7472.583} C_VEL
LIN {X 0,Y 467.741,Z 147.724,A -85,B 0,C 180,E1 -7476.037,E2 -7476.037} C_VEL
LIN {X 0,Y 467.679,Z 147.729,A -85,B 0,C 180,E1 -7478.643,E2 -7478.643} C_VEL
LIN {X 0,Y 467.652,Z 147.734,A -85,B 0,C 180,E1 -7482.145,E2 -7482.145} C_VEL
LIN {X 0,Y 467.635,Z 147.737,A -85,B 0,C 180,E1 -7485.695,E2 -7485.695} C_VEL
LIN {X 0,Y 467.614,Z 147.737,A -85,B 0,C 180,E1 -7488.765,E2 -7488.765} C_VEL
LIN {X 0,Y 467.577,Z 147.745,A -85,B 0,C 180,E1 -7491.268,E2 -7491.268} C_VEL
LIN {X 0,Y 467.569,Z 147.742,A -85,B 0,C 180,E1 -7493.943,E2 -7493.943} C_VEL
LIN {X 0,Y 467.612,Z 147.737,A -85,B 0,C 180,E1 -7496.8,E2 -7496.8} C_VEL
LIN {X 0,Y 467.584,Z 147.734,A -85,B 0,C 180,E1 -7499.736,E2 -7499.736} C_VEL
LIN {X 0,Y 467.579,Z 147.742,A -85,B 0,C 180,E1 -7502.758,E2 -7502.758} C_VEL
LIN {X 0,Y 467.551,Z 147.737,A -85,B 0,C 180,E1 -7505.889,E2 -7505.889} C_VEL
LIN {X 0,Y 467.578,Z 147.739,A -85,B 0,C 180,E1 -7509.145,E2 -7509.145} C_VEL
LIN {X 0,Y 467.581,Z 147.717,A -85,B 0,C 180,E1 -7512.567,E2 -7512.567} C_VEL
LIN {X 0,Y 467.566,Z 147.743,A -85,B 0,C 180,E1 -7515.053,E2 -7515.053} C_VEL
LIN {X 0,Y 467.583,Z 147.737,A -85,B 0,C 180,E1 -7517.44,E2 -7517.44} C_VEL
LIN {X 0,Y 467.577,Z 147.744,A -85,B 0,C 180,E1 -7520.855,E2 -7520.855} C_VEL
LIN {X 0,Y 467.558,Z 147.743,A -85,B 0,C 180,E1 -7524.26,E2 -7524.26} C_VEL
LIN {X 0,Y 467.577,Z 147.737,A -85,B 0,C 180,E1 -7527.321,E2 -7527.321} C_VEL
LIN {X 0,Y 467.565,Z 147.738,A -85,B 0,C 180,E1 -7530.668,E2 -7530.668} C_VEL
LIN {X 0,Y 467.622,Z 147.723,A -85,B 0,C 180,E1 -7533.201,E2 -7533.201} C_VEL
LIN {X 0,Y 467.588,Z 147.741,A -85,B 0,C 180,E1 -7536.468,E2 -7536.468} C_VEL
LIN {X 0,Y 467.618,Z 147.73,A -85,B 0,C 180,E1 -7539.778,E2 -7539.778} C_VEL
LIN {X 0,Y 467.604,Z 147.733,A -85,B 0,C 180,E1 -7542.507,E2 -7542.507} C_VEL
LIN {X 0,Y 467.602,Z 147.735,A -85,B 0,C 180,E1 -7545.197,E2 -7545.197} C_VEL
LIN {X 0,Y 467.651,Z 147.728,A -85,B 0,C 180,E1 -7547.855,E2 -7547.855} C_VEL
LIN {X 0,Y 467.677,Z 147.714,A -85,B 0,C 180,E1 -7551.358,E2 -7551.358} C_VEL
LIN {X 0,Y 467.739,Z 147.723,A -85,B 0,C 180,E1 -7553.963,E2 -7553.963} C_VEL
LIN {X 0,Y 467.856,Z 147.705,A -85,B 0,C 180,E1 -7557.418,E2 -7557.418} C_VEL
LIN {X 0,Y 467.878,Z 147.689,A -85,B 0,C 180,E1 -7560,E2 -7560} C_VEL
LIN {X 0,Y 467.856,Z 147.699,A -85,B 0,C 180,E1 -7562.583,E2 -7562.583} C_VEL
LIN {X 0,Y 467.74,Z 147.717,A -85,B 0,C 180,E1 -7566.038,E2 -7566.038} C_VEL
LIN {X 0,Y 467.678,Z 147.715,A -85,B 0,C 180,E1 -7568.643,E2 -7568.643} C_VEL
LIN {X 0,Y 467.653,Z 147.724,A -85,B 0,C 180,E1 -7572.146,E2 -7572.146} C_VEL
LIN {X 0,Y 467.636,Z 147.728,A -85,B 0,C 180,E1 -7575.696,E2 -7575.696} C_VEL
LIN {X 0,Y 467.615,Z 147.722,A -85,B 0,C 180,E1 -7578.765,E2 -7578.765} C_VEL
LIN {X 0,Y 467.578,Z 147.741,A -85,B 0,C 180,E1 -7581.269,E2 -7581.269} C_VEL
LIN {X 0,Y 467.569,Z 147.737,A -85,B 0,C 180,E1 -7583.944,E2 -7583.944} C_VEL
LIN {X 0,Y 467.614,Z 147.727,A -85,B 0,C 180,E1 -7586.801,E2 -7586.801} C_VEL
LIN {X 0,Y 467.552,Z 147.74,A -85,B 0,C 180,E1 -7589.739,E2 -7589.739} C_VEL
LIN {X 0,Y 467.582,Z 147.737,A -85,B 0,C 180,E1 -7592.759,E2 -7592.759} C_VEL
LIN {X 0,Y 467.553,Z 147.738,A -85,B 0,C 180,E1 -7595.89,E2 -7595.89} C_VEL
LIN {X 0,Y 467.559,Z 147.737,A -85,B 0,C 180,E1 -7599.148,E2 -7599.148} C_VEL
LIN {X 0,Y 467.586,Z 147.743,A -85,B 0,C 180,E1 -7602.568,E2 -7602.568} C_VEL
LIN {X 0,Y 467.566,Z 147.74,A -85,B 0,C 180,E1 -7605.053,E2 -7605.053} C_VEL
LIN {X 0,Y 467.589,Z 147.737,A -85,B 0,C 180,E1 -7607.441,E2 -7607.441} C_VEL
LIN {X 0,Y 467.583,Z 147.737,A -85,B 0,C 180,E1 -7610.856,E2 -7610.856} C_VEL
LIN {X 0,Y 467.561,Z 147.737,A -85,B 0,C 180,E1 -7614.261,E2 -7614.261} C_VEL
LIN {X 0,Y 467.583,Z 147.738,A -85,B 0,C 180,E1 -7617.321,E2 -7617.321} C_VEL
LIN {X 0,Y 467.57,Z 147.741,A -85,B 0,C 180,E1 -7620.668,E2 -7620.668} C_VEL
LIN {X 0,Y 467.685,Z 147.899,A -85,B 0,C 180,E1 -7622.503,E2 -7622.503} C_VEL
LIN {X 0,Y 469.402,Z 157.924,A -85,B 0,C 180,E1 -7624.978,E2 -7624.978} C_VEL
LIN {X 0,Y 468.913,Z 169.202,A -85,B 0,C 180,E1 -7627.531,E2 -7627.531} C_VEL
LIN {X 0,Y 468.326,Z 182.648,A -85,B 0,C 180,E1 -7630.495,E2 -7630.495} C_VEL
LIN {X 0,Y 467.906,Z 192.708,A -85,B 0,C 180,E1 -7632.744,E2 -7632.744} C_VEL
LIN {X 0,Y 467.927,Z 194.014,A -85,B 0,C 180,E1 -7632.969,E2 -7632.969} C_VEL
LIN {X 0,Y 471.219,Z 214.049,A -85,B 0,C 180,E1 -7633.427,E2 -7633.427} C_VEL
LIN {X 0,Y 470.582,Z 298.661,A -85,B 0,C 180,E1 -7634.739,E2 -7634.739} C_VEL
LIN {X 0,Y 470.321,Z 309.431,A -85,B 0,C 180,E1 -7635.007,E2 -7635.007} C_VEL
LIN {X 0,Y 470.056,Z 318.533,A -85,B 0,C 180,E1 -7635.331,E2 -7635.331} C_VEL
LIN {X 0,Y 469.626,Z 328.896,A -85,B 0,C 180,E1 -7635.815,E2 -7635.815} C_VEL
LIN {X 0,Y 469.236,Z 338.031,A -85,B 0,C 180,E1 -7636.356,E2 -7636.356} C_VEL
LIN {X 0,Y 468.78,Z 347.362,A -85,B 0,C 180,E1 -7637.031,E2 -7637.031} C_VEL
LIN {X 0,Y 468.485,Z 355.058,A -85,B 0,C 180,E1 -7637.698,E2 -7637.698} C_VEL
LIN {X 0,Y 468.11,Z 363.158,A -85,B 0,C 180,E1 -7638.526,E2 -7638.526} C_VEL
LIN {X 0,Y 467.736,Z 370.378,A -85,B 0,C 180,E1 -7639.394,E2 -7639.394} C_VEL
LIN {X 0,Y 467.448,Z 376.58,A -85,B 0,C 180,E1 -7640.262,E2 -7640.262} C_VEL
LIN {X 0,Y 467.156,Z 383.118,A -85,B 0,C 180,E1 -7641.348,E2 -7641.348} C_VEL
LIN {X 0,Y 466.977,Z 387.619,A -85,B 0,C 180,E1 -7642.215,E2 -7642.215} C_VEL
LIN {X 0,Y 466.793,Z 393.274,A -85,B 0,C 180,E1 -7643.563,E2 -7643.563} C_VEL
LIN {X 0,Y 466.735,Z 397.431,A -85,B 0,C 180,E1 -7644.817,E2 -7644.817} C_VEL
LIN {X 0,Y 466.647,Z 399.794,A -85,B 0,C 180,E1 -7645.681,E2 -7645.681} C_VEL
LIN {X 0,Y 466.689,Z 401.591,A -85,B 0,C 180,E1 -7646.547,E2 -7646.547} C_VEL
LIN {X 0,Y 466.608,Z 404.03,A -85,B 0,C 180,E1 -7648.274,E2 -7648.274} C_VEL
LIN {X 0,Y 466.62,Z 404.618,A -85,B 0,C 180,E1 -7649.137,E2 -7649.137} C_VEL
LIN {X 0,Y 466.62,Z 404.618,A -85,B 0,C 180,E1 -7650.863,E2 -7650.863} C_VEL
LIN {X 0,Y 466.608,Z 404.03,A -85,B 0,C 180,E1 -7651.726,E2 -7651.726} C_VEL
LIN {X 0,Y 466.689,Z 401.591,A -85,B 0,C 180,E1 -7653.453,E2 -7653.453} C_VEL
LIN {X 0,Y 466.69,Z 398.646,A -85,B 0,C 180,E1 -7654.751,E2 -7654.751} C_VEL
LIN {X 0,Y 466.744,Z 394.661,A -85,B 0,C 180,E1 -7656.05,E2 -7656.05} C_VEL
LIN {X 0,Y 466.868,Z 389.533,A -85,B 0,C 180,E1 -7657.351,E2 -7657.351} C_VEL
LIN {X 0,Y 467.107,Z 384.273,A -85,B 0,C 180,E1 -7658.435,E2 -7658.435} C_VEL
LIN {X 0,Y 467.362,Z 377.956,A -85,B 0,C 180,E1 -7659.521,E2 -7659.521} C_VEL
LIN {X 0,Y 467.614,Z 372.004,A -85,B 0,C 180,E1 -7660.39,E2 -7660.39} C_VEL
LIN {X 0,Y 468.003,Z 365.077,A -85,B 0,C 180,E1 -7661.257,E2 -7661.257} C_VEL
LIN {X 0,Y 468.412,Z 356.897,A -85,B 0,C 180,E1 -7662.125,E2 -7662.125} C_VEL
LIN {X 0,Y 468.769,Z 348.096,A -85,B 0,C 180,E1 -7662.909,E2 -7662.909} C_VEL
LIN {X 0,Y 469.172,Z 339.664,A -85,B 0,C 180,E1 -7663.536,E2 -7663.536} C_VEL
LIN {X 0,Y 469.546,Z 329.902,A -85,B 0,C 180,E1 -7664.132,E2 -7664.132} C_VEL
LIN {X 0,Y 469.992,Z 319.82,A -85,B 0,C 180,E1 -7664.616,E2 -7664.616} C_VEL
LIN {X 0,Y 470.287,Z 310.305,A -85,B 0,C 180,E1 -7664.966,E2 -7664.966} C_VEL
LIN {X 0,Y 470.503,Z 301.324,A -85,B 0,C 180,E1 -7665.208,E2 -7665.208} C_VEL
LIN {X 0,Y 470.808,Z 277.147,A -85,B 0,C 180,E1 -7665.608,E2 -7665.608} C_VEL
LIN {X 0,Y 471.032,Z 211.95,A -85,B 0,C 180,E1 -7666.613,E2 -7666.613} C_VEL
LIN {X 0,Y 467.943,Z 194.12,A -85,B 0,C 180,E1 -7667.023,E2 -7667.023} C_VEL
LIN {X 0,Y 467.912,Z 192.613,A -85,B 0,C 180,E1 -7667.278,E2 -7667.278} C_VEL
LIN {X 0,Y 468.522,Z 179.758,A -85,B 0,C 180,E1 -7670.182,E2 -7670.182} C_VEL
LIN {X 0,Y 469.266,Z 163.082,A -85,B 0,C 180,E1 -7673.851,E2 -7673.851} C_VEL
LIN {X 0,Y 469.336,Z 156.902,A -85,B 0,C 180,E1 -7675.262,E2 -7675.262} C_VEL
LIN {X 0,Y 467.676,Z 147.778,A -85,B 0,C 180,E1 -7677.548,E2 -7677.548} C_VEL
LIN {X 0,Y 467.57,Z 147.743,A -85,B 0,C 180,E1 -7681.044,E2 -7681.044} C_VEL
LIN {X 0,Y 467.589,Z 147.738,A -85,B 0,C 180,E1 -7684.242,E2 -7684.242} C_VEL
LIN {X 0,Y 467.549,Z 147.743,A -85,B 0,C 180,E1 -7687.186,E2 -7687.186} C_VEL
LIN {X 0,Y 467.578,Z 147.728,A -85,B 0,C 180,E1 -7690.264,E2 -7690.264} C_VEL
LIN {X 0,Y 467.587,Z 147.737,A -85,B 0,C 180,E1 -7692.566,E2 -7692.566} C_VEL
LIN {X 0,Y 467.566,Z 147.74,A -85,B 0,C 180,E1 -7695.052,E2 -7695.052} C_VEL
LIN {X 0,Y 467.589,Z 147.744,A -85,B 0,C 180,E1 -7697.439,E2 -7697.439} C_VEL
LIN {X 0,Y 467.559,Z 147.737,A -85,B 0,C 180,E1 -7700.852,E2 -7700.852} C_VEL
LIN {X 0,Y 467.559,Z 147.737,A -85,B 0,C 180,E1 -7704.26,E2 -7704.26} C_VEL
LIN {X 0,Y 467.581,Z 147.739,A -85,B 0,C 180,E1 -7707.32,E2 -7707.32} C_VEL
LIN {X 0,Y 467.568,Z 147.74,A -85,B 0,C 180,E1 -7710.667,E2 -7710.667} C_VEL
LIN {X 0,Y 467.614,Z 147.727,A -85,B 0,C 180,E1 -7713.199,E2 -7713.199} C_VEL
LIN {X 0,Y 467.59,Z 147.736,A -85,B 0,C 180,E1 -7716.468,E2 -7716.468} C_VEL
LIN {X 0,Y 467.62,Z 147.724,A -85,B 0,C 180,E1 -7719.777,E2 -7719.777} C_VEL
LIN {X 0,Y 467.606,Z 147.724,A -85,B 0,C 180,E1 -7722.506,E2 -7722.506} C_VEL
LIN {X 0,Y 467.604,Z 147.736,A -85,B 0,C 180,E1 -7725.196,E2 -7725.196} C_VEL
LIN {X 0,Y 467.653,Z 147.724,A -85,B 0,C 180,E1 -7727.854,E2 -7727.854} C_VEL
LIN {X 0,Y 467.678,Z 147.715,A -85,B 0,C 180,E1 -7731.357,E2 -7731.357} C_VEL
LIN {X 0,Y 467.74,Z 147.717,A -85,B 0,C 180,E1 -7733.962,E2 -7733.962} C_VEL
LIN {X 0,Y 467.856,Z 147.699,A -85,B 0,C 180,E1 -7737.417,E2 -7737.417} C_VEL
LIN {X 0,Y 467.878,Z 147.689,A -85,B 0,C 180,E1 -7740,E2 -7740} C_VEL
LIN {X 0,Y 467.856,Z 147.705,A -85,B 0,C 180,E1 -7742.582,E2 -7742.582} C_VEL
LIN {X 0,Y 467.739,Z 147.723,A -85,B 0,C 180,E1 -7746.037,E2 -7746.037} C_VEL
LIN {X 0,Y 467.677,Z 147.714,A -85,B 0,C 180,E1 -7748.642,E2 -7748.642} C_VEL
LIN {X 0,Y 467.651,Z 147.728,A -85,B 0,C 180,E1 -7752.145,E2 -7752.145} C_VEL
LIN {X 0,Y 467.634,Z 147.735,A -85,B 0,C 180,E1 -7755.695,E2 -7755.695} C_VEL
LIN {X 0,Y 467.612,Z 147.719,A -85,B 0,C 180,E1 -7758.764,E2 -7758.764} C_VEL
LIN {X 0,Y 467.576,Z 147.734,A -85,B 0,C 180,E1 -7761.268,E2 -7761.268} C_VEL
LIN {X 0,Y 467.569,Z 147.743,A -85,B 0,C 180,E1 -7763.943,E2 -7763.943} C_VEL
LIN {X 0,Y 467.622,Z 147.723,A -85,B 0,C 180,E1 -7766.799,E2 -7766.799} C_VEL
LIN {X 0,Y 467.575,Z 147.744,A -85,B 0,C 180,E1 -7769.736,E2 -7769.736} C_VEL
LIN {X 0,Y 467.579,Z 147.737,A -85,B 0,C 180,E1 -7772.758,E2 -7772.758} C_VEL
LIN {X 0,Y 467.552,Z 147.742,A -85,B 0,C 180,E1 -7775.889,E2 -7775.889} C_VEL
LIN {X 0,Y 467.577,Z 147.744,A -85,B 0,C 180,E1 -7779.145,E2 -7779.145} C_VEL
LIN {X 0,Y 467.581,Z 147.737,A -85,B 0,C 180,E1 -7782.567,E2 -7782.567} C_VEL
LIN {X 0,Y 467.566,Z 147.741,A -85,B 0,C 180,E1 -7785.053,E2 -7785.053} C_VEL
LIN {X 0,Y 467.584,Z 147.716,A -85,B 0,C 180,E1 -7787.44,E2 -7787.44} C_VEL
LIN {X 0,Y 467.578,Z 147.739,A -85,B 0,C 180,E1 -7790.855,E2 -7790.855} C_VEL
LIN {X 0,Y 467.558,Z 147.736,A -85,B 0,C 180,E1 -7794.26,E2 -7794.26} C_VEL
LIN {X 0,Y 467.578,Z 147.741,A -85,B 0,C 180,E1 -7797.321,E2 -7797.321} C_VEL
LIN {X 0,Y 467.573,Z 147.734,A -85,B 0,C 180,E1 -7800.666,E2 -7800.666} C_VEL
LIN {X 0,Y 467.612,Z 147.737,A -85,B 0,C 180,E1 -7803.2,E2 -7803.2} C_VEL
LIN {X 0,Y 467.589,Z 147.743,A -85,B 0,C 180,E1 -7806.468,E2 -7806.468} C_VEL
LIN {X 0,Y 467.62,Z 147.736,A -85,B 0,C 180,E1 -7809.777,E2 -7809.777} C_VEL
LIN {X 0,Y 467.605,Z 147.741,A -85,B 0,C 180,E1 -7812.507,E2 -7812.507} C_VEL
LIN {X 0,Y 467.593,Z 147.739,A -85,B 0,C 180,E1 -7815.413,E2 -7815.413} C_VEL
LIN {X 0,Y 466.923,Z 147.826,A -85,B 0,C 180,E1 -7816.132,E2 -7816.132} C_VEL
LIN {X 0,Y 464.08,Z 148.177,A -85,B 0,C 180,E1 -7817.301,E2 -7817.301} C_VEL
LIN {X 0,Y 461.682,Z 148.479,A -85,B 0,C 180,E1 -7818.243,E2 -7818.243} C_VEL
LIN {X 0,Y 460.656,Z 148.604,A -85,B 0,C 180,E1 -7818.971,E2 -7818.971} C_VEL
LIN {X 0,Y 460.574,Z 148.613,A -85,B 0,C 180,E1 -7819.217,E2 -7819.217} C_VEL
LIN {X 0,Y 460.717,Z 148.599,A -85,B 0,C 180,E1 -7822.538,E2 -7822.538} C_VEL
LIN {X 0,Y 460.695,Z 148.6,A -85,B 0,C 180,E1 -7824.748,E2 -7824.748} C_VEL
LIN {X 0,Y 460.822,Z 148.584,A -85,B 0,C 180,E1 -7827.378,E2 -7827.378} C_VEL
LIN {X 0,Y 460.85,Z 148.583,A -85,B 0,C 180,E1 -7830,E2 -7830} C_VEL
LIN {X 0,Y 460.822,Z 148.584,A -85,B 0,C 180,E1 -7832.622,E2 -7832.622} C_VEL
LIN {X 0,Y 460.707,Z 148.601,A -85,B 0,C 180,E1 -7836.13,E2 -7836.13} C_VEL
LIN {X 0,Y 460.626,Z 148.608,A -85,B 0,C 180,E1 -7838.776,E2 -7838.776} C_VEL
LIN {X 0,Y 460.609,Z 148.61,A -85,B 0,C 180,E1 -7842.445,E2 -7842.445} C_VEL
LIN {X 0,Y 460.596,Z 148.613,A -85,B 0,C 180,E1 -7845.997,E2 -7845.997} C_VEL
LIN {X 0,Y 460.567,Z 148.615,A -85,B 0,C 180,E1 -7848.902,E2 -7848.902} C_VEL
LIN {X 0,Y 460.512,Z 148.625,A -85,B 0,C 180,E1 -7851.486,E2 -7851.486} C_VEL
LIN {X 0,Y 460.538,Z 148.616,A -85,B 0,C 180,E1 -7854.332,E2 -7854.332} C_VEL
LIN {X 0,Y 460.576,Z 148.617,A -85,B 0,C 180,E1 -7857.243,E2 -7857.243} C_VEL
LIN {X 0,Y 460.527,Z 148.612,A -85,B 0,C 180,E1 -7860.238,E2 -7860.238} C_VEL
LIN {X 0,Y 460.525,Z 148.611,A -85,B 0,C 180,E1 -7863.325,E2 -7863.325} C_VEL
LIN {X 0,Y 460.473,Z 148.62,A -85,B 0,C 180,E1 -7866.529,E2 -7866.529} C_VEL
LIN {X 0,Y 460.54,Z 148.619,A -85,B 0,C 180,E1 -7868.898,E2 -7868.898} C_VEL
LIN {X 0,Y 460.517,Z 148.593,A -85,B 0,C 180,E1 -7872.181,E2 -7872.181} C_VEL
LIN {X 0,Y 460.515,Z 148.618,A -85,B 0,C 180,E1 -7875.412,E2 -7875.412} C_VEL
LIN {X 0,Y 460.53,Z 148.618,A -85,B 0,C 180,E1 -7878.397,E2 -7878.397} C_VEL
LIN {X 0,Y 460.521,Z 148.618,A -85,B 0,C 180,E1 -7881.267,E2 -7881.267} C_VEL
LIN {X 0,Y 460.508,Z 148.616,A -85,B 0,C 180,E1 -7884.555,E2 -7884.555} C_VEL
LIN {X 0,Y 460.527,Z 148.615,A -85,B 0,C 180,E1 -7887.716,E2 -7887.716} C_VEL
LIN {X 0,Y 460.535,Z 148.613,A -85,B 0,C 180,E1 -7890.769,E2 -7890.769} C_VEL
LIN {X 0,Y 460.563,Z 148.603,A -85,B 0,C 180,E1 -7893.735,E2 -7893.735} C_VEL
LIN {X 0,Y 460.542,Z 148.617,A -85,B 0,C 180,E1 -7896.624,E2 -7896.624} C_VEL
LIN {X 0,Y 460.546,Z 148.609,A -85,B 0,C 180,E1 -7899.453,E2 -7899.453} C_VEL
LIN {X 0,Y 460.555,Z 148.608,A -85,B 0,C 180,E1 -7902.231,E2 -7902.231} C_VEL
LIN {X 0,Y 460.561,Z 148.612,A -85,B 0,C 180,E1 -7904.965,E2 -7904.965} C_VEL
LIN {X 0,Y 460.607,Z 148.597,A -85,B 0,C 180,E1 -7908.56,E2 -7908.56} C_VEL
LIN {X 0,Y 460.691,Z 148.595,A -85,B 0,C 180,E1 -7912.109,E2 -7912.109} C_VEL
LIN {X 0,Y 460.693,Z 148.595,A -85,B 0,C 180,E1 -7914.749,E2 -7914.749} C_VEL
LIN {X 0,Y 460.821,Z 148.581,A -85,B 0,C 180,E1 -7917.378,E2 -7917.378} C_VEL
LIN {X 0,Y 460.849,Z 148.564,A -85,B 0,C 180,E1 -7920,E2 -7920} C_VEL
LIN {X 0,Y 460.797,Z 148.578,A -85,B 0,C 180,E1 -7922.623,E2 -7922.623} C_VEL
LIN {X 0,Y 460.706,Z 148.592,A -85,B 0,C 180,E1 -7926.13,E2 -7926.13} C_VEL
LIN {X 0,Y 460.625,Z 148.594,A -85,B 0,C 180,E1 -7928.777,E2 -7928.777} C_VEL
LIN {X 0,Y 460.61,Z 148.601,A -85,B 0,C 180,E1 -7932.445,E2 -7932.445} C_VEL
LIN {X 0,Y 460.597,Z 148.603,A -85,B 0,C 180,E1 -7935.998,E2 -7935.998} C_VEL
LIN {X 0,Y 460.568,Z 148.599,A -85,B 0,C 180,E1 -7938.902,E2 -7938.902} C_VEL
LIN {X 0,Y 460.513,Z 148.619,A -85,B 0,C 180,E1 -7941.486,E2 -7941.486} C_VEL
LIN {X 0,Y 460.539,Z 148.614,A -85,B 0,C 180,E1 -7944.333,E2 -7944.333} C_VEL
LIN {X 0,Y 460.571,Z 148.604,A -85,B 0,C 180,E1 -7947.244,E2 -7947.244} C_VEL
LIN {X 0,Y 460.509,Z 148.619,A -85,B 0,C 180,E1 -7950.241,E2 -7950.241} C_VEL
LIN {X 0,Y 460.528,Z 148.609,A -85,B 0,C 180,E1 -7953.325,E2 -7953.325} C_VEL
LIN {X 0,Y 460.475,Z 148.626,A -85,B 0,C 180,E1 -7956.53,E2 -7956.53} C_VEL
LIN {X 0,Y 460.524,Z 148.612,A -85,B 0,C 180,E1 -7959.864,E2 -7959.864} C_VEL
LIN {X 0,Y 460.511,Z 148.62,A -85,B 0,C 180,E1 -7962.901,E2 -7962.901} C_VEL
LIN {X 0,Y 460.509,Z 148.619,A -85,B 0,C 180,E1 -7965.831,E2 -7965.831} C_VEL
LIN {X 0,Y 460.531,Z 148.606,A -85,B 0,C 180,E1 -7968.989,E2 -7968.989} C_VEL
LIN {X 0,Y 460.527,Z 148.615,A -85,B 0,C 180,E1 -7971.268,E2 -7971.268} C_VEL
LIN {X 0,Y 460.511,Z 148.615,A -85,B 0,C 180,E1 -7974.555,E2 -7974.555} C_VEL
LIN {X 0,Y 460.533,Z 148.615,A -85,B 0,C 180,E1 -7977.716,E2 -7977.716} C_VEL
LIN {X 0,Y 460.541,Z 148.617,A -85,B 0,C 180,E1 -7980.769,E2 -7980.769} C_VEL
LIN {X 0,Y 460.644,Z 148.794,A -85,B 0,C 180,E1 -7982.293,E2 -7982.293} C_VEL
LIN {X 0,Y 462.408,Z 158.809,A -85,B 0,C 180,E1 -7984.814,E2 -7984.814} C_VEL
LIN {X 0,Y 462.093,Z 166.964,A -85,B 0,C 180,E1 -7986.707,E2 -7986.707} C_VEL
LIN {X 0,Y 461.507,Z 180.417,A -85,B 0,C 180,E1 -7989.73,E2 -7989.73} C_VEL
LIN {X 0,Y 460.931,Z 192.521,A -85,B 0,C 180,E1 -7992.474,E2 -7992.474} C_VEL
LIN {X 0,Y 460.912,Z 193.825,A -85,B 0,C 180,E1 -7992.702,E2 -7992.702} C_VEL
LIN {X 0,Y 464.362,Z 213.856,A -85,B 0,C 180,E1 -7993.175,E2 -7993.175} C_VEL
LIN {X 0,Y 463.736,Z 298.47,A -85,B 0,C 180,E1 -7994.508,E2 -7994.508} C_VEL
LIN {X 0,Y 463.478,Z 309.239,A -85,B 0,C 180,E1 -7994.781,E2 -7994.781} C_VEL
LIN {X 0,Y 463.181,Z 318.341,A -85,B 0,C 180,E1 -7995.108,E2 -7995.108} C_VEL
LIN {X 0,Y 462.741,Z 328.704,A -85,B 0,C 180,E1 -7995.6,E2 -7995.6} C_VEL
LIN {X 0,Y 462.331,Z 337.839,A -85,B 0,C 180,E1 -7996.148,E2 -7996.148} C_VEL
LIN {X 0,Y 461.857,Z 346.837,A -85,B 0,C 180,E1 -7996.806,E2 -7996.806} C_VEL
LIN {X 0,Y 461.514,Z 355.055,A -85,B 0,C 180,E1 -7997.528,E2 -7997.528} C_VEL
LIN {X 0,Y 461.108,Z 362.965,A -85,B 0,C 180,E1 -7998.349,E2 -7998.349} C_VEL
LIN {X 0,Y 460.727,Z 370.185,A -85,B 0,C 180,E1 -7999.23,E2 -7999.23} C_VEL
LIN {X 0,Y 460.436,Z 376.388,A -85,B 0,C 180,E1 -8000.112,E2 -8000.112} C_VEL
LIN {X 0,Y 460.117,Z 382.925,A -85,B 0,C 180,E1 -8001.214,E2 -8001.214} C_VEL
LIN {X 0,Y 459.899,Z 387.426,A -85,B 0,C 180,E1 -8002.095,E2 -8002.095} C_VEL
LIN {X 0,Y 459.736,Z 392.409,A -85,B 0,C 180,E1 -8003.273,E2 -8003.273} C_VEL
LIN {X 0,Y 459.648,Z 397.239,A -85,B 0,C 180,E1 -8004.736,E2 -8004.736} C_VEL
LIN {X 0,Y 459.565,Z 399.602,A -85,B 0,C 180,E1 -8005.615,E2 -8005.615} C_VEL
LIN {X 0,Y 459.584,Z 401.399,A -85,B 0,C 180,E1 -8006.493,E2 -8006.493} C_VEL
LIN {X 0,Y 459.52,Z 403.839,A -85,B 0,C 180,E1 -8008.247,E2 -8008.247} C_VEL
LIN {X 0,Y 459.523,Z 404.427,A -85,B 0,C 180,E1 -8009.124,E2 -8009.124} C_VEL
LIN {X 0,Y 459.523,Z 404.427,A -85,B 0,C 180,E1 -8010.876,E2 -8010.876} C_VEL
LIN {X 0,Y 459.52,Z 403.839,A -85,B 0,C 180,E1 -8011.753,E2 -8011.753} C_VEL
LIN {X 0,Y 459.584,Z 401.399,A -85,B 0,C 180,E1 -8013.507,E2 -8013.507} C_VEL
LIN {X 0,Y 459.618,Z 398.454,A -85,B 0,C 180,E1 -8014.824,E2 -8014.824} C_VEL
LIN {X 0,Y 459.655,Z 394.468,A -85,B 0,C 180,E1 -8016.144,E2 -8016.144} C_VEL
LIN {X 0,Y 459.813,Z 389.341,A -85,B 0,C 180,E1 -8017.465,E2 -8017.465} C_VEL
LIN {X 0,Y 460.044,Z 384.08,A -85,B 0,C 180,E1 -8018.566,E2 -8018.566} C_VEL
LIN {X 0,Y 460.329,Z 377.764,A -85,B 0,C 180,E1 -8019.668,E2 -8019.668} C_VEL
LIN {X 0,Y 460.599,Z 371.811,A -85,B 0,C 180,E1 -8020.55,E2 -8020.55} C_VEL
LIN {X 0,Y 461.017,Z 364.885,A -85,B 0,C 180,E1 -8021.43,E2 -8021.43} C_VEL
LIN {X 0,Y 461.434,Z 356.704,A -85,B 0,C 180,E1 -8022.312,E2 -8022.312} C_VEL
LIN {X 0,Y 461.82,Z 347.942,A -85,B 0,C 180,E1 -8023.104,E2 -8023.104} C_VEL
LIN {X 0,Y 462.241,Z 339.471,A -85,B 0,C 180,E1 -8023.743,E2 -8023.743} C_VEL
LIN {X 0,Y 462.67,Z 329.711,A -85,B 0,C 180,E1 -8024.347,E2 -8024.347} C_VEL
LIN {X 0,Y 463.14,Z 319.629,A -85,B 0,C 180,E1 -8024.837,E2 -8024.837} C_VEL
LIN {X 0,Y 463.451,Z 310.114,A -85,B 0,C 180,E1 -8025.192,E2 -8025.192} C_VEL
LIN {X 0,Y 463.66,Z 301.132,A -85,B 0,C 180,E1 -8025.438,E2 -8025.438} C_VEL
LIN {X 0,Y 463.982,Z 277.031,A -85,B 0,C 180,E1 -8025.842,E2 -8025.842} C_VEL
LIN {X 0,Y 464.278,Z 213.059,A -85,B 0,C 180,E1 -8026.841,E2 -8026.841} C_VEL
LIN {X 0,Y 460.928,Z 194.218,A -85,B 0,C 180,E1 -8027.275,E2 -8027.275} C_VEL
LIN {X 0,Y 460.919,Z 192.851,A -85,B 0,C 180,E1 -8027.446,E2 -8027.446} C_VEL
LIN {X 0,Y 461.52,Z 180.617,A -85,B 0,C 180,E1 -8030.269,E2 -8030.269} C_VEL
LIN {X 0,Y 462.256,Z 165.078,A -85,B 0,C 180,E1 -8033.751,E2 -8033.751} C_VEL
LIN {X 0,Y 462.434,Z 158.81,A -85,B 0,C 180,E1 -8035.185,E2 -8035.185} C_VEL
LIN {X 0,Y 460.622,Z 148.678,A -85,B 0,C 180,E1 -8037.755,E2 -8037.755} C_VEL
LIN {X 0,Y 460.523,Z 148.623,A -85,B 0,C 180,E1 -8041.282,E2 -8041.282} C_VEL
LIN {X 0,Y 460.533,Z 148.615,A -85,B 0,C 180,E1 -8044.505,E2 -8044.505} C_VEL
LIN {X 0,Y 460.528,Z 148.622,A -85,B 0,C 180,E1 -8047.62,E2 -8047.62} C_VEL
LIN {X 0,Y 460.542,Z 148.604,A -85,B 0,C 180,E1 -8050.269,E2 -8050.269} C_VEL
LIN {X 0,Y 460.499,Z 148.625,A -85,B 0,C 180,E1 -8053.375,E2 -8053.375} C_VEL
LIN {X 0,Y 460.496,Z 148.62,A -85,B 0,C 180,E1 -8056.624,E2 -8056.624} C_VEL
LIN {X 0,Y 460.538,Z 148.613,A -85,B 0,C 180,E1 -8059.73,E2 -8059.73} C_VEL
LIN {X 0,Y 460.498,Z 148.62,A -85,B 0,C 180,E1 -8062.523,E2 -8062.523} C_VEL
LIN {X 0,Y 460.545,Z 148.608,A -85,B 0,C 180,E1 -8065.623,E2 -8065.623} C_VEL
LIN {X 0,Y 460.536,Z 148.617,A -85,B 0,C 180,E1 -8068.744,E2 -8068.744} C_VEL
LIN {X 0,Y 460.58,Z 148.602,A -85,B 0,C 180,E1 -8072.253,E2 -8072.253} C_VEL
LIN {X 0,Y 460.557,Z 148.607,A -85,B 0,C 180,E1 -8074.705,E2 -8074.705} C_VEL
LIN {X 0,Y 460.508,Z 148.618,A -85,B 0,C 180,E1 -8077.571,E2 -8077.571} C_VEL
LIN {X 0,Y 460.566,Z 148.604,A -85,B 0,C 180,E1 -8080.384,E2 -8080.384} C_VEL
LIN {X 0,Y 460.563,Z 148.611,A -85,B 0,C 180,E1 -8083.146,E2 -8083.146} C_VEL
LIN {X 0,Y 460.555,Z 148.611,A -85,B 0,C 180,E1 -8085.868,E2 -8085.868} C_VEL
LIN {X 0,Y 460.607,Z 148.602,A -85,B 0,C 180,E1 -8088.559,E2 -8088.559} C_VEL
LIN {X 0,Y 460.692,Z 148.587,A -85,B 0,C 180,E1 -8092.108,E2 -8092.108} C_VEL
LIN {X 0,Y 460.694,Z 148.6,A -85,B 0,C 180,E1 -8094.748,E2 -8094.748} C_VEL
LIN {X 0,Y 460.797,Z 148.578,A -85,B 0,C 180,E1 -8097.377,E2 -8097.377} C_VEL
LIN {X 0,Y 460.849,Z 148.564,A -85,B 0,C 180,E1 -8100,E2 -8100} C_VEL
LIN {X 0,Y 460.821,Z 148.581,A -85,B 0,C 180,E1 -8102.622,E2 -8102.622} C_VEL
LIN {X 0,Y 460.705,Z 148.6,A -85,B 0,C 180,E1 -8106.129,E2 -8106.129} C_VEL
LIN {X 0,Y 460.624,Z 148.591,A -85,B 0,C 180,E1 -8108.776,E2 -8108.776} C_VEL
LIN {X 0,Y 460.609,Z 148.607,A -85,B 0,C 180,E1 -8112.445,E2 -8112.445} C_VEL
LIN {X 0,Y 460.595,Z 148.611,A -85,B 0,C 180,E1 -8115.997,E2 -8115.997} C_VEL
LIN {X 0,Y 460.566,Z 148.596,A -85,B 0,C 180,E1 -8118.901,E2 -8118.901} C_VEL
LIN {X 0,Y 460.511,Z 148.616,A -85,B 0,C 180,E1 -8121.485,E2 -8121.485} C_VEL
LIN {X 0,Y 460.538,Z 148.614,A -85,B 0,C 180,E1 -8124.332,E2 -8124.332} C_VEL
LIN {X 0,Y 460.579,Z 148.602,A -85,B 0,C 180,E1 -8127.243,E2 -8127.243} C_VEL
LIN {X 0,Y 460.517,Z 148.619,A -85,B 0,C 180,E1 -8130.239,E2 -8130.239} C_VEL
LIN {X 0,Y 460.524,Z 148.617,A -85,B 0,C 180,E1 -8133.325,E2 -8133.325} C_VEL
LIN {X 0,Y 460.474,Z 148.622,A -85,B 0,C 180,E1 -8136.529,E2 -8136.529} C_VEL
LIN {X 0,Y 460.54,Z 148.617,A -85,B 0,C 180,E1 -8138.898,E2 -8138.898} C_VEL
LIN {X 0,Y 460.519,Z 148.616,A -85,B 0,C 180,E1 -8142.181,E2 -8142.181} C_VEL
LIN {X 0,Y 460.515,Z 148.613,A -85,B 0,C 180,E1 -8145.412,E2 -8145.412} C_VEL
LIN {X 0,Y 460.527,Z 148.593,A -85,B 0,C 180,E1 -8148.397,E2 -8148.397} C_VEL
LIN {X 0,Y 460.522,Z 148.623,A -85,B 0,C 180,E1 -8151.267,E2 -8151.267} C_VEL
LIN {X 0,Y 460.509,Z 148.612,A -85,B 0,C 180,E1 -8154.555,E2 -8154.555} C_VEL
LIN {X 0,Y 460.529,Z 148.617,A -85,B 0,C 180,E1 -8157.716,E2 -8157.716} C_VEL
LIN {X 0,Y 460.542,Z 148.609,A -85,B 0,C 180,E1 -8160.77,E2 -8160.77} C_VEL
LIN {X 0,Y 460.559,Z 148.614,A -85,B 0,C 180,E1 -8163.735,E2 -8163.735} C_VEL
LIN {X 0,Y 460.542,Z 148.621,A -85,B 0,C 180,E1 -8166.624,E2 -8166.624} C_VEL
LIN {X 0,Y 460.548,Z 148.616,A -85,B 0,C 180,E1 -8169.453,E2 -8169.453} C_VEL
LIN {X 0,Y 460.556,Z 148.619,A -85,B 0,C 180,E1 -8172.23,E2 -8172.23} C_VEL
LIN {X 0,Y 460.562,Z 148.616,A -85,B 0,C 180,E1 -8174.965,E2 -8174.965} C_VEL
LIN {X 0,Y 460.608,Z 148.612,A -85,B 0,C 180,E1 -8178.559,E2 -8178.559} C_VEL
LIN {X 0,Y 460.574,Z 148.613,A -85,B 0,C 180,E1 -8179.217,E2 -8179.217} C_VEL
LIN {X 0,Y 459.919,Z 148.698,A -85,B 0,C 180,E1 -8179.947,E2 -8179.947} C_VEL
LIN {X 0,Y 457.102,Z 149.049,A -85,B 0,C 180,E1 -8181.134,E2 -8181.134} C_VEL
LIN {X 0,Y 454.723,Z 149.346,A -85,B 0,C 180,E1 -8182.091,E2 -8182.091} C_VEL
LIN {X 0,Y 453.711,Z 149.47,A -85,B 0,C 180,E1 -8182.83,E2 -8182.83} C_VEL
LIN {X 0,Y 453.633,Z 149.479,A -85,B 0,C 180,E1 -8183.08,E2 -8183.08} C_VEL
LIN {X 0,Y 453.668,Z 149.476,A -85,B 0,C 180,E1 -8184.667,E2 -8184.667} C_VEL
LIN {X 0,Y 453.762,Z 149.463,A -85,B 0,C 180,E1 -8187.337,E2 -8187.337} C_VEL
LIN {X 0,Y 453.821,Z 149.459,A -85,B 0,C 180,E1 -8190,E2 -8190} C_VEL
LIN {X 0,Y 453.762,Z 149.463,A -85,B 0,C 180,E1 -8192.663,E2 -8192.663} C_VEL
LIN {X 0,Y 453.675,Z 149.476,A -85,B 0,C 180,E1 -8196.225,E2 -8196.225} C_VEL
LIN {X 0,Y 453.589,Z 149.485,A -85,B 0,C 180,E1 -8198.913,E2 -8198.913} C_VEL
LIN {X 0,Y 453.56,Z 149.488,A -85,B 0,C 180,E1 -8202.529,E2 -8202.529} C_VEL
LIN {X 0,Y 453.541,Z 149.491,A -85,B 0,C 180,E1 -8206.196,E2 -8206.196} C_VEL
LIN {X 0,Y 453.517,Z 149.495,A -85,B 0,C 180,E1 -8209.041,E2 -8209.041} C_VEL
LIN {X 0,Y 453.473,Z 149.5,A -85,B 0,C 180,E1 -8211.836,E2 -8211.836} C_VEL
LIN {X 0,Y 453.51,Z 149.493,A -85,B 0,C 180,E1 -8214.734,E2 -8214.734} C_VEL
LIN {X 0,Y 453.534,Z 149.487,A -85,B 0,C 180,E1 -8217.961,E2 -8217.961} C_VEL
LIN {X 0,Y 453.48,Z 149.493,A -85,B 0,C 180,E1 -8220.759,E2 -8220.759} C_VEL
LIN {X 0,Y 453.473,Z 149.484,A -85,B 0,C 180,E1 -8223.913,E2 -8223.913} C_VEL
LIN {X 0,Y 453.465,Z 149.502,A -85,B 0,C 180,E1 -8227.188,E2 -8227.188} C_VEL
LIN {X 0,Y 453.485,Z 149.49,A -85,B 0,C 180,E1 -8229.45,E2 -8229.45} C_VEL
LIN {X 0,Y 453.471,Z 149.47,A -85,B 0,C 180,E1 -8231.935,E2 -8231.935} C_VEL
LIN {X 0,Y 453.486,Z 149.494,A -85,B 0,C 180,E1 -8235.47,E2 -8235.47} C_VEL
LIN {X 0,Y 453.476,Z 149.495,A -85,B 0,C 180,E1 -8238.21,E2 -8238.21} C_VEL
LIN {X 0,Y 453.505,Z 149.494,A -85,B 0,C 180,E1 -8240.791,E2 -8240.791} C_VEL
LIN {X 0,Y 453.452,Z 149.497,A -85,B 0,C 180,E1 -8243.918,E2 -8243.918} C_VEL
LIN {X 0,Y 453.478,Z 149.494,A -85,B 0,C 180,E1 -8247.151,E2 -8247.151} C_VEL
LIN {X 0,Y 453.492,Z 149.497,A -85,B 0,C 180,E1 -8250.27,E2 -8250.27} C_VEL
LIN {X 0,Y 453.509,Z 149.48,A -85,B 0,C 180,E1 -8253.295,E2 -8253.295} C_VEL
LIN {X 0,Y 453.499,Z 149.498,A -85,B 0,C 180,E1 -8256.239,E2 -8256.239} C_VEL
LIN {X 0,Y 453.477,Z 149.488,A -85,B 0,C 180,E1 -8259.118,E2 -8259.118} C_VEL
LIN {X 0,Y 453.507,Z 149.48,A -85,B 0,C 180,E1 -8261.945,E2 -8261.945} C_VEL
LIN {X 0,Y 453.535,Z 149.488,A -85,B 0,C 180,E1 -8264.727,E2 -8264.727} C_VEL
LIN {X 0,Y 453.555,Z 149.476,A -85,B 0,C 180,E1 -8268.379,E2 -8268.379} C_VEL
LIN {X 0,Y 453.648,Z 149.47,A -85,B 0,C 180,E1 -8271.986,E2 -8271.986} C_VEL
LIN {X 0,Y 453.667,Z 149.471,A -85,B 0,C 180,E1 -8274.667,E2 -8274.667} C_VEL
LIN {X 0,Y 453.761,Z 149.46,A -85,B 0,C 180,E1 -8277.337,E2 -8277.337} C_VEL
LIN {X 0,Y 453.819,Z 149.438,A -85,B 0,C 180,E1 -8280,E2 -8280} C_VEL
LIN {X 0,Y 453.741,Z 149.457,A -85,B 0,C 180,E1 -8282.664,E2 -8282.664} C_VEL
LIN {X 0,Y 453.674,Z 149.468,A -85,B 0,C 180,E1 -8286.226,E2 -8286.226} C_VEL
LIN {X 0,Y 453.589,Z 149.471,A -85,B 0,C 180,E1 -8288.914,E2 -8288.914} C_VEL
LIN {X 0,Y 453.561,Z 149.479,A -85,B 0,C 180,E1 -8292.529,E2 -8292.529} C_VEL
LIN {X 0,Y 453.542,Z 149.482,A -85,B 0,C 180,E1 -8296.196,E2 -8296.196} C_VEL
LIN {X 0,Y 453.517,Z 149.477,A -85,B 0,C 180,E1 -8299.041,E2 -8299.041} C_VEL
LIN {X 0,Y 453.474,Z 149.493,A -85,B 0,C 180,E1 -8301.837,E2 -8301.837} C_VEL
LIN {X 0,Y 453.511,Z 149.493,A -85,B 0,C 180,E1 -8304.735,E2 -8304.735} C_VEL
LIN {X 0,Y 453.53,Z 149.479,A -85,B 0,C 180,E1 -8307.96,E2 -8307.96} C_VEL
LIN {X 0,Y 453.465,Z 149.496,A -85,B 0,C 180,E1 -8311.526,E2 -8311.526} C_VEL
LIN {X 0,Y 453.486,Z 149.489,A -85,B 0,C 180,E1 -8314.778,E2 -8314.778} C_VEL
LIN {X 0,Y 453.459,Z 149.501,A -85,B 0,C 180,E1 -8318.313,E2 -8318.313} C_VEL
LIN {X 0,Y 453.493,Z 149.492,A -85,B 0,C 180,E1 -8320.61,E2 -8320.61} C_VEL
LIN {X 0,Y 453.452,Z 149.497,A -85,B 0,C 180,E1 -8323.244,E2 -8323.244} C_VEL
LIN {X 0,Y 453.463,Z 149.496,A -85,B 0,C 180,E1 -8325.779,E2 -8325.779} C_VEL
LIN {X 0,Y 453.479,Z 149.493,A -85,B 0,C 180,E1 -8328.21,E2 -8328.21} C_VEL
LIN {X 0,Y 453.511,Z 149.489,A -85,B 0,C 180,E1 -8330.791,E2 -8330.791} C_VEL
LIN {X 0,Y 453.455,Z 149.496,A -85,B 0,C 180,E1 -8333.918,E2 -8333.918} C_VEL
LIN {X 0,Y 453.484,Z 149.494,A -85,B 0,C 180,E1 -8337.152,E2 -8337.152} C_VEL
LIN {X 0,Y 453.476,Z 149.495,A -85,B 0,C 180,E1 -8340.269,E2 -8340.269} C_VEL
LIN {X 0,Y 453.594,Z 149.701,A -85,B 0,C 180,E1 -8342.08,E2 -8342.08} C_VEL
LIN {X 0,Y 455.389,Z 159.694,A -85,B 0,C 180,E1 -8344.643,E2 -8344.643} C_VEL
LIN {X 0,Y 455.294,Z 165.185,A -85,B 0,C 180,E1 -8345.962,E2 -8345.962} C_VEL
LIN {X 0,Y 454.556,Z 180.253,A -85,B 0,C 180,E1 -8349.406,E2 -8349.406} C_VEL
LIN {X 0,Y 453.959,Z 192.332,A -85,B 0,C 180,E1 -8352.196,E2 -8352.196} C_VEL
LIN {X 0,Y 453.921,Z 193.637,A -85,B 0,C 180,E1 -8352.427,E2 -8352.427} C_VEL
LIN {X 0,Y 457.591,Z 215.059,A -85,B 0,C 180,E1 -8352.941,E2 -8352.941} C_VEL
LIN {X 0,Y 456.895,Z 298.278,A -85,B 0,C 180,E1 -8354.27,E2 -8354.27} C_VEL
LIN {X 0,Y 456.634,Z 308.173,A -85,B 0,C 180,E1 -8354.518,E2 -8354.518} C_VEL
LIN {X 0,Y 456.317,Z 318.149,A -85,B 0,C 180,E1 -8354.879,E2 -8354.879} C_VEL
LIN {X 0,Y 455.933,Z 327.506,A -85,B 0,C 180,E1 -8355.323,E2 -8355.323} C_VEL
LIN {X 0,Y 455.42,Z 337.647,A -85,B 0,C 180,E1 -8355.933,E2 -8355.933} C_VEL
LIN {X 0,Y 454.924,Z 346.644,A -85,B 0,C 180,E1 -8356.601,E2 -8356.601} C_VEL
LIN {X 0,Y 454.547,Z 355.063,A -85,B 0,C 180,E1 -8357.354,E2 -8357.354} C_VEL
LIN {X 0,Y 454.111,Z 362.772,A -85,B 0,C 180,E1 -8358.167,E2 -8358.167} C_VEL
LIN {X 0,Y 453.697,Z 369.992,A -85,B 0,C 180,E1 -8359.061,E2 -8359.061} C_VEL
LIN {X 0,Y 453.384,Z 376.195,A -85,B 0,C 180,E1 -8359.957,E2 -8359.957} C_VEL
LIN {X 0,Y 453.044,Z 382.732,A -85,B 0,C 180,E1 -8361.076,E2 -8361.076} C_VEL
LIN {X 0,Y 452.847,Z 387.234,A -85,B 0,C 180,E1 -8361.971,E2 -8361.971} C_VEL
LIN {X 0,Y 452.64,Z 392.725,A -85,B 0,C 180,E1 -8363.313,E2 -8363.313} C_VEL
LIN {X 0,Y 452.562,Z 397.047,A -85,B 0,C 180,E1 -8364.654,E2 -8364.654} C_VEL
LIN {X 0,Y 452.487,Z 399.41,A -85,B 0,C 180,E1 -8365.546,E2 -8365.546} C_VEL
LIN {X 0,Y 452.48,Z 401.207,A -85,B 0,C 180,E1 -8366.438,E2 -8366.438} C_VEL
LIN {X 0,Y 452.437,Z 403.648,A -85,B 0,C 180,E1 -8368.22,E2 -8368.22} C_VEL
LIN {X 0,Y 452.43,Z 404.235,A -85,B 0,C 180,E1 -8369.11,E2 -8369.11} C_VEL
LIN {X 0,Y 452.43,Z 404.235,A -85,B 0,C 180,E1 -8370.89,E2 -8370.89} C_VEL
LIN {X 0,Y 452.437,Z 403.648,A -85,B 0,C 180,E1 -8371.78,E2 -8371.78} C_VEL
LIN {X 0,Y 452.48,Z 401.207,A -85,B 0,C 180,E1 -8373.562,E2 -8373.562} C_VEL
LIN {X 0,Y 452.546,Z 398.263,A -85,B 0,C 180,E1 -8374.9,E2 -8374.9} C_VEL
LIN {X 0,Y 452.585,Z 394.276,A -85,B 0,C 180,E1 -8376.24,E2 -8376.24} C_VEL
LIN {X 0,Y 452.738,Z 389.148,A -85,B 0,C 180,E1 -8377.582,E2 -8377.582} C_VEL
LIN {X 0,Y 453.004,Z 383.888,A -85,B 0,C 180,E1 -8378.7,E2 -8378.7} C_VEL
LIN {X 0,Y 453.314,Z 377.571,A -85,B 0,C 180,E1 -8379.819,E2 -8379.819} C_VEL
LIN {X 0,Y 453.592,Z 371.619,A -85,B 0,C 180,E1 -8380.715,E2 -8380.715} C_VEL
LIN {X 0,Y 454.032,Z 364.693,A -85,B 0,C 180,E1 -8381.609,E2 -8381.609} C_VEL
LIN {X 0,Y 454.467,Z 356.511,A -85,B 0,C 180,E1 -8382.503,E2 -8382.503} C_VEL
LIN {X 0,Y 454.855,Z 348.574,A -85,B 0,C 180,E1 -8383.239,E2 -8383.239} C_VEL
LIN {X 0,Y 455.324,Z 339.279,A -85,B 0,C 180,E1 -8383.956,E2 -8383.956} C_VEL
LIN {X 0,Y 455.793,Z 329.519,A -85,B 0,C 180,E1 -8384.568,E2 -8384.568} C_VEL
LIN {X 0,Y 456.196,Z 320.725,A -85,B 0,C 180,E1 -8385.011,E2 -8385.011} C_VEL
LIN {X 0,Y 456.56,Z 310.796,A -85,B 0,C 180,E1 -8385.399,E2 -8385.399} C_VEL
